LIN {X 0,Y 305.408,Z 165.44,A -85,B 0,C 180,E1 -15880.59,E2 -15880.59} C_VEL
LIN {X 0,Y 305.42,Z 165.439,A -85,B 0,C 180,E1 -15883.657,E2 -15883.657} C_VEL
LIN {X 0,Y 305.434,Z 165.438,A -85,B 0,C 180,E1 -15887.419,E2 -15887.419} C_VEL
LIN {X 0,Y 305.46,Z 165.434,A -85,B 0,C 180,E1 -15891.596,E2 -15891.596} C_VEL
LIN {X 0,Y 305.462,Z 165.438,A -85,B 0,C 180,E1 -15894.887,E2 -15894.887} C_VEL
LIN {X 0,Y 305.446,Z 165.457,A -85,B 0,C 180,E1 -15898.262,E2 -15898.262} C_VEL
LIN {X 0,Y 308.056,Z 177.958,A -85,B 0,C 180,E1 -15902.116,E2 -15902.116} C_VEL
LIN {X 0,Y 309.424,Z 185.81,A -85,B 0,C 180,E1 -15904.434,E2 -15904.434} C_VEL
LIN {X 0,Y 309.211,Z 188.563,A -85,B 0,C 180,E1 -15905.192,E2 -15905.192} C_VEL
LIN {X 0,Y 314.924,Z 228.362,A -85,B 0,C 180,E1 -15906.653,E2 -15906.653} C_VEL
LIN {X 0,Y 313.069,Z 297.497,A -85,B 0,C 180,E1 -15908.433,E2 -15908.433} C_VEL
LIN {X 0,Y 312.295,Z 311.547,A -85,B 0,C 180,E1 -15909.068,E2 -15909.068} C_VEL
LIN {X 0,Y 311.224,Z 323.574,A -85,B 0,C 180,E1 -15909.857,E2 -15909.857} C_VEL
LIN {X 0,Y 310.032,Z 336.146,A -85,B 0,C 180,E1 -15910.982,E2 -15910.982} C_VEL
LIN {X 0,Y 308.666,Z 347.394,A -85,B 0,C 180,E1 -15912.27,E2 -15912.27} C_VEL
LIN {X 0,Y 307.454,Z 358.217,A -85,B 0,C 180,E1 -15913.852,E2 -15913.852} C_VEL
LIN {X 0,Y 306.459,Z 366.753,A -85,B 0,C 180,E1 -15915.389,E2 -15915.389} C_VEL
LIN {X 0,Y 305.37,Z 375.712,A -85,B 0,C 180,E1 -15917.371,E2 -15917.371} C_VEL
LIN {X 0,Y 304.591,Z 382.844,A -85,B 0,C 180,E1 -15919.363,E2 -15919.363} C_VEL
LIN {X 0,Y 304.06,Z 388.526,A -85,B 0,C 180,E1 -15921.359,E2 -15921.359} C_VEL
LIN {X 0,Y 303.758,Z 392.963,A -85,B 0,C 180,E1 -15923.357,E2 -15923.357} C_VEL
LIN {X 0,Y 303.668,Z 395.298,A -85,B 0,C 180,E1 -15924.688,E2 -15924.688} C_VEL
LIN {X 0,Y 303.634,Z 397.179,A -85,B 0,C 180,E1 -15926.018,E2 -15926.018} C_VEL
LIN {X 0,Y 303.608,Z 398.571,A -85,B 0,C 180,E1 -15927.346,E2 -15927.346} C_VEL
LIN {X 0,Y 303.576,Z 399.548,A -85,B 0,C 180,E1 -15928.673,E2 -15928.673} C_VEL
LIN {X 0,Y 303.605,Z 400.123,A -85,B 0,C 180,E1 -15930,E2 -15930} C_VEL
LIN {X 0,Y 303.566,Z 400.276,A -85,B 0,C 180,E1 -15931.326,E2 -15931.326} C_VEL
LIN {X 0,Y 303.602,Z 399.989,A -85,B 0,C 180,E1 -15932.653,E2 -15932.653} C_VEL
LIN {X 0,Y 303.592,Z 399.306,A -85,B 0,C 180,E1 -15933.982,E2 -15933.982} C_VEL
LIN {X 0,Y 303.627,Z 398.001,A -85,B 0,C 180,E1 -15935.544,E2 -15935.544} C_VEL
LIN {X 0,Y 304.004,Z 394.748,A -85,B 0,C 180,E1 -15937.973,E2 -15937.973} C_VEL
LIN {X 0,Y 304.538,Z 390.959,A -85,B 0,C 180,E1 -15939.967,E2 -15939.967} C_VEL
LIN {X 0,Y 305.368,Z 386.046,A -85,B 0,C 180,E1 -15941.954,E2 -15941.954} C_VEL
LIN {X 0,Y 306.544,Z 379.882,A -85,B 0,C 180,E1 -15943.929,E2 -15943.929} C_VEL
LIN {X 0,Y 308.159,Z 372.25,A -85,B 0,C 180,E1 -15945.883,E2 -15945.883} C_VEL
LIN {X 0,Y 309.396,Z 364.671,A -85,B 0,C 180,E1 -15947.481,E2 -15947.481} C_VEL
LIN {X 0,Y 311.169,Z 355.095,A -85,B 0,C 180,E1 -15949.116,E2 -15949.116} C_VEL
LIN {X 0,Y 313.044,Z 344.695,A -85,B 0,C 180,E1 -15950.535,E2 -15950.535} C_VEL
LIN {X 0,Y 314.841,Z 333.237,A -85,B 0,C 180,E1 -15951.783,E2 -15951.783} C_VEL
LIN {X 0,Y 316.432,Z 321.299,A -85,B 0,C 180,E1 -15952.785,E2 -15952.785} C_VEL
LIN {X 0,Y 317.803,Z 308.332,A -85,B 0,C 180,E1 -15953.586,E2 -15953.586} C_VEL
LIN {X 0,Y 318.869,Z 294.721,A -85,B 0,C 180,E1 -15954.149,E2 -15954.149} C_VEL
LIN {X 0,Y 321.21,Z 229.462,A -85,B 0,C 180,E1 -15955.868,E2 -15955.868} C_VEL
LIN {X 0,Y 318.444,Z 211.613,A -85,B 0,C 180,E1 -15956.729,E2 -15956.729} C_VEL
LIN {X 0,Y 315.326,Z 197.331,A -85,B 0,C 180,E1 -15957.545,E2 -15957.545} C_VEL
LIN {X 0,Y 310.558,Z 186.54,A -85,B 0,C 180,E1 -15958.519,E2 -15958.519} C_VEL
LIN {X 0,Y 308.899,Z 178.602,A -85,B 0,C 180,E1 -15961.194,E2 -15961.194} C_VEL
LIN {X 0,Y 306.662,Z 169.805,A -85,B 0,C 180,E1 -15964.407,E2 -15964.407} C_VEL
LIN {X 0,Y 305.483,Z 165.436,A -85,B 0,C 180,E1 -15966.139,E2 -15966.139} C_VEL
LIN {X 0,Y 305.408,Z 165.445,A -85,B 0,C 180,E1 -15970.114,E2 -15970.114} C_VEL
LIN {X 0,Y 305.418,Z 165.446,A -85,B 0,C 180,E1 -15973.655,E2 -15973.655} C_VEL
LIN {X 0,Y 305.431,Z 165.435,A -85,B 0,C 180,E1 -15977.418,E2 -15977.418} C_VEL
LIN {X 0,Y 305.438,Z 165.439,A -85,B 0,C 180,E1 -15981.591,E2 -15981.591} C_VEL
LIN {X 0,Y 305.458,Z 165.437,A -85,B 0,C 180,E1 -15984.886,E2 -15984.886} C_VEL
LIN {X 0,Y 305.438,Z 165.438,A -85,B 0,C 180,E1 -15988.358,E2 -15988.358} C_VEL
LIN {X 0,Y 305.459,Z 165.432,A -85,B 0,C 180,E1 -15991.107,E2 -15991.107} C_VEL
LIN {X 0,Y 305.474,Z 165.424,A -85,B 0,C 180,E1 -15994.078,E2 -15994.078} C_VEL
LIN {X 0,Y 305.452,Z 165.431,A -85,B 0,C 180,E1 -15998.399,E2 -15998.399} C_VEL
LIN {X 0,Y 305.494,Z 165.421,A -85,B 0,C 180,E1 -16001.211,E2 -16001.211} C_VEL
LIN {X 0,Y 305.573,Z 165.414,A -85,B 0,C 180,E1 -16005.345,E2 -16005.345} C_VEL
LIN {X 0,Y 305.617,Z 165.413,A -85,B 0,C 180,E1 -16009.398,E2 -16009.398} C_VEL
LIN {X 0,Y 305.74,Z 165.394,A -85,B 0,C 180,E1 -16012.072,E2 -16012.072} C_VEL
LIN {X 0,Y 305.648,Z 165.405,A -85,B 0,C 180,E1 -16014.722,E2 -16014.722} C_VEL
LIN {X 0,Y 305.928,Z 165.375,A -85,B 0,C 180,E1 -16018.683,E2 -16018.683} C_VEL
LIN {X 0,Y 305.928,Z 165.374,A -85,B 0,C 180,E1 -16021.316,E2 -16021.316} C_VEL
LIN {X 0,Y 305.777,Z 165.398,A -85,B 0,C 180,E1 -16026.598,E2 -16026.598} C_VEL
LIN {X 0,Y 305.688,Z 165.41,A -85,B 0,C 180,E1 -16029.261,E2 -16029.261} C_VEL
LIN {X 0,Y 305.626,Z 165.55,A -85,B 0,C 180,E1 -16031.944,E2 -16031.944} C_VEL
LIN {X 0,Y 307.793,Z 173.872,A -85,B 0,C 180,E1 -16035.181,E2 -16035.181} C_VEL
LIN {X 0,Y 315.177,Z 188.448,A -85,B 0,C 180,E1 -16036.629,E2 -16036.629} C_VEL
LIN {X 0,Y 321.1,Z 202.216,A -85,B 0,C 180,E1 -16037.761,E2 -16037.761} C_VEL
LIN {X 0,Y 322.097,Z 207.438,A -85,B 0,C 180,E1 -16038.033,E2 -16038.033} C_VEL
LIN {X 0,Y 319.132,Z 281.719,A -85,B 0,C 180,E1 -16039.983,E2 -16039.983} C_VEL
LIN {X 0,Y 318.191,Z 294.602,A -85,B 0,C 180,E1 -16040.555,E2 -16040.555} C_VEL
LIN {X 0,Y 317.006,Z 307.445,A -85,B 0,C 180,E1 -16041.39,E2 -16041.39} C_VEL
LIN {X 0,Y 315.544,Z 319.205,A -85,B 0,C 180,E1 -16042.421,E2 -16042.421} C_VEL
LIN {X 0,Y 314.01,Z 329.384,A -85,B 0,C 180,E1 -16043.549,E2 -16043.549} C_VEL
LIN {X 0,Y 312.228,Z 339.663,A -85,B 0,C 180,E1 -16044.963,E2 -16044.963} C_VEL
LIN {X 0,Y 310.555,Z 348.97,A -85,B 0,C 180,E1 -16046.559,E2 -16046.559} C_VEL
LIN {X 0,Y 308.735,Z 358.223,A -85,B 0,C 180,E1 -16048.557,E2 -16048.557} C_VEL
LIN {X 0,Y 307.18,Z 365.75,A -85,B 0,C 180,E1 -16050.601,E2 -16050.601} C_VEL
LIN {X 0,Y 305.96,Z 371.708,A -85,B 0,C 180,E1 -16052.669,E2 -16052.669} C_VEL
LIN {X 0,Y 304.868,Z 377.163,A -85,B 0,C 180,E1 -16055.191,E2 -16055.191} C_VEL
LIN {X 0,Y 304.311,Z 379.879,A -85,B 0,C 180,E1 -16056.902,E2 -16056.902} C_VEL
LIN {X 0,Y 303.863,Z 381.909,A -85,B 0,C 180,E1 -16058.643,E2 -16058.643} C_VEL
LIN {X 0,Y 303.576,Z 383.185,A -85,B 0,C 180,E1 -16060.407,E2 -16060.407} C_VEL
LIN {X 0,Y 303.368,Z 383.757,A -85,B 0,C 180,E1 -16062.208,E2 -16062.208} C_VEL
LIN {X 0,Y 303.301,Z 383.572,A -85,B 0,C 180,E1 -16064.085,E2 -16064.085} C_VEL
LIN {X 0,Y 303.365,Z 382.564,A -85,B 0,C 180,E1 -16065.974,E2 -16065.974} C_VEL
LIN {X 0,Y 303.533,Z 380.734,A -85,B 0,C 180,E1 -16067.821,E2 -16067.821} C_VEL
LIN {X 0,Y 303.8,Z 377.908,A -85,B 0,C 180,E1 -16069.765,E2 -16069.765} C_VEL
LIN {X 0,Y 304.26,Z 373.976,A -85,B 0,C 180,E1 -16071.753,E2 -16071.753} C_VEL
LIN {X 0,Y 304.811,Z 368.708,A -85,B 0,C 180,E1 -16073.802,E2 -16073.802} C_VEL
LIN {X 0,Y 305.595,Z 361.864,A -85,B 0,C 180,E1 -16075.884,E2 -16075.884} C_VEL
LIN {X 0,Y 306.663,Z 353.083,A -85,B 0,C 180,E1 -16077.989,E2 -16077.989} C_VEL
LIN {X 0,Y 307.765,Z 344.443,A -85,B 0,C 180,E1 -16079.654,E2 -16079.654} C_VEL
LIN {X 0,Y 308.949,Z 333.974,A -85,B 0,C 180,E1 -16081.279,E2 -16081.279} C_VEL
LIN {X 0,Y 310.201,Z 322.827,A -85,B 0,C 180,E1 -16082.658,E2 -16082.658} C_VEL
LIN {X 0,Y 311.315,Z 310.616,A -85,B 0,C 180,E1 -16083.842,E2 -16083.842} C_VEL
LIN {X 0,Y 312.329,Z 297.638,A -85,B 0,C 180,E1 -16084.778,E2 -16084.778} C_VEL
LIN {X 0,Y 313.018,Z 284.837,A -85,B 0,C 180,E1 -16085.436,E2 -16085.436} C_VEL
LIN {X 0,Y 313.553,Z 268.917,A -85,B 0,C 180,E1 -16085.921,E2 -16085.921} C_VEL
LIN {X 0,Y 315.327,Z 203.407,A -85,B 0,C 180,E1 -16087.573,E2 -16087.573} C_VEL
LIN {X 0,Y 312.589,Z 189.103,A -85,B 0,C 180,E1 -16088.139,E2 -16088.139} C_VEL
LIN {X 0,Y 306.9,Z 172.553,A -85,B 0,C 180,E1 -16088.991,E2 -16088.991} C_VEL
LIN {X 0,Y 305.545,Z 165.426,A -85,B 0,C 180,E1 -16091.389,E2 -16091.389} C_VEL
LIN {X 0,Y 305.575,Z 165.42,A -85,B 0,C 180,E1 -16095.346,E2 -16095.346} C_VEL
LIN {X 0,Y 305.619,Z 165.413,A -85,B 0,C 180,E1 -16099.399,E2 -16099.399} C_VEL
LIN {X 0,Y 305.743,Z 165.401,A -85,B 0,C 180,E1 -16102.073,E2 -16102.073} C_VEL
LIN {X 0,Y 305.653,Z 165.41,A -85,B 0,C 180,E1 -16104.723,E2 -16104.723} C_VEL
LIN {X 0,Y 305.931,Z 165.376,A -85,B 0,C 180,E1 -16108.684,E2 -16108.684} C_VEL
LIN {X 0,Y 305.93,Z 165.375,A -85,B 0,C 180,E1 -16111.317,E2 -16111.317} C_VEL
LIN {X 0,Y 305.781,Z 165.394,A -85,B 0,C 180,E1 -16116.599,E2 -16116.599} C_VEL
LIN {X 0,Y 305.691,Z 165.405,A -85,B 0,C 180,E1 -16119.261,E2 -16119.261} C_VEL
LIN {X 0,Y 305.566,Z 165.421,A -85,B 0,C 180,E1 -16123.297,E2 -16123.297} C_VEL
LIN {X 0,Y 305.508,Z 165.429,A -85,B 0,C 180,E1 -16126.025,E2 -16126.025} C_VEL
LIN {X 0,Y 305.472,Z 165.432,A -85,B 0,C 180,E1 -16130.188,E2 -16130.188} C_VEL
LIN {X 0,Y 305.435,Z 165.436,A -85,B 0,C 180,E1 -16134.467,E2 -16134.467} C_VEL
LIN {X 0,Y 305.437,Z 165.44,A -85,B 0,C 180,E1 -16137.399,E2 -16137.399} C_VEL
LIN {X 0,Y 305.413,Z 165.438,A -85,B 0,C 180,E1 -16140.414,E2 -16140.414} C_VEL
LIN {X 0,Y 305.461,Z 165.432,A -85,B 0,C 180,E1 -16144.078,E2 -16144.078} C_VEL
LIN {X 0,Y 305.449,Z 165.435,A -85,B 0,C 180,E1 -16146.743,E2 -16146.743} C_VEL
LIN {X 0,Y 305.405,Z 165.44,A -85,B 0,C 180,E1 -16150.59,E2 -16150.59} C_VEL
LIN {X 0,Y 305.416,Z 165.437,A -85,B 0,C 180,E1 -16153.656,E2 -16153.656} C_VEL
LIN {X 0,Y 305.43,Z 165.438,A -85,B 0,C 180,E1 -16157.419,E2 -16157.419} C_VEL
LIN {X 0,Y 305.455,Z 165.434,A -85,B 0,C 180,E1 -16161.595,E2 -16161.595} C_VEL
LIN {X 0,Y 305.439,Z 165.435,A -85,B 0,C 180,E1 -16163.128,E2 -16163.128} C_VEL
LIN {X 0,Y 304.826,Z 165.519,A -85,B 0,C 180,E1 -16164.228,E2 -16164.228} C_VEL
LIN {X 0,Y 301.99,Z 165.879,A -85,B 0,C 180,E1 -16166.019,E2 -16166.019} C_VEL
LIN {X 0,Y 299.537,Z 166.181,A -85,B 0,C 180,E1 -16167.471,E2 -16167.471} C_VEL
LIN {X 0,Y 298.46,Z 166.308,A -85,B 0,C 180,E1 -16168.596,E2 -16168.596} C_VEL
LIN {X 0,Y 298.363,Z 166.317,A -85,B 0,C 180,E1 -16168.978,E2 -16168.978} C_VEL
LIN {X 0,Y 298.404,Z 166.311,A -85,B 0,C 180,E1 -16171.899,E2 -16171.899} C_VEL
LIN {X 0,Y 298.408,Z 166.314,A -85,B 0,C 180,E1 -16174.918,E2 -16174.918} C_VEL
LIN {X 0,Y 298.386,Z 166.313,A -85,B 0,C 180,E1 -16177.862,E2 -16177.862} C_VEL
LIN {X 0,Y 298.448,Z 166.304,A -85,B 0,C 180,E1 -16180.751,E2 -16180.751} C_VEL
LIN {X 0,Y 298.506,Z 166.298,A -85,B 0,C 180,E1 -16184.991,E2 -16184.991} C_VEL
LIN {X 0,Y 298.576,Z 166.29,A -85,B 0,C 180,E1 -16189.147,E2 -16189.147} C_VEL
LIN {X 0,Y 298.68,Z 166.278,A -85,B 0,C 180,E1 -16191.884,E2 -16191.884} C_VEL
LIN {X 0,Y 298.62,Z 166.282,A -85,B 0,C 180,E1 -16194.599,E2 -16194.599} C_VEL
LIN {X 0,Y 298.897,Z 166.25,A -85,B 0,C 180,E1 -16198.653,E2 -16198.653} C_VEL
LIN {X 0,Y 298.897,Z 166.25,A -85,B 0,C 180,E1 -16201.348,E2 -16201.348} C_VEL
LIN {X 0,Y 298.728,Z 166.268,A -85,B 0,C 180,E1 -16206.756,E2 -16206.756} C_VEL
LIN {X 0,Y 298.614,Z 166.287,A -85,B 0,C 180,E1 -16209.483,E2 -16209.483} C_VEL
LIN {X 0,Y 298.519,Z 166.301,A -85,B 0,C 180,E1 -16213.617,E2 -16213.617} C_VEL
LIN {X 0,Y 298.443,Z 166.305,A -85,B 0,C 180,E1 -16216.415,E2 -16216.415} C_VEL
LIN {X 0,Y 298.426,Z 166.314,A -85,B 0,C 180,E1 -16219.61,E2 -16219.61} C_VEL
LIN {X 0,Y 298.379,Z 166.318,A -85,B 0,C 180,E1 -16223.605,E2 -16223.605} C_VEL
LIN {X 0,Y 298.399,Z 166.313,A -85,B 0,C 180,E1 -16226.584,E2 -16226.584} C_VEL
LIN {X 0,Y 298.355,Z 166.321,A -85,B 0,C 180,E1 -16229.649,E2 -16229.649} C_VEL
LIN {X 0,Y 298.391,Z 166.312,A -85,B 0,C 180,E1 -16232.801,E2 -16232.801} C_VEL
LIN {X 0,Y 298.426,Z 166.31,A -85,B 0,C 180,E1 -16236.803,E2 -16236.803} C_VEL
LIN {X 0,Y 298.373,Z 166.318,A -85,B 0,C 180,E1 -16239.493,E2 -16239.493} C_VEL
LIN {X 0,Y 298.369,Z 166.321,A -85,B 0,C 180,E1 -16243.098,E2 -16243.098} C_VEL
LIN {X 0,Y 298.37,Z 166.321,A -85,B 0,C 180,E1 -16246.915,E2 -16246.915} C_VEL
LIN {X 0,Y 298.385,Z 166.319,A -85,B 0,C 180,E1 -16251.012,E2 -16251.012} C_VEL
LIN {X 0,Y 298.405,Z 166.313,A -85,B 0,C 180,E1 -16253.929,E2 -16253.929} C_VEL
LIN {X 0,Y 298.421,Z 166.42,A -85,B 0,C 180,E1 -16257.932,E2 -16257.932} C_VEL
LIN {X 0,Y 300.947,Z 178.583,A -85,B 0,C 180,E1 -16261.778,E2 -16261.778} C_VEL
LIN {X 0,Y 302.396,Z 186.453,A -85,B 0,C 180,E1 -16264.164,E2 -16264.164} C_VEL
LIN {X 0,Y 302.387,Z 188.388,A -85,B 0,C 180,E1 -16264.72,E2 -16264.72} C_VEL
LIN {X 0,Y 308.176,Z 228.777,A -85,B 0,C 180,E1 -16266.25,E2 -16266.25} C_VEL
LIN {X 0,Y 306.271,Z 297.409,A -85,B 0,C 180,E1 -16268.062,E2 -16268.062} C_VEL
LIN {X 0,Y 305.454,Z 311.406,A -85,B 0,C 180,E1 -16268.709,E2 -16268.709} C_VEL
LIN {X 0,Y 304.33,Z 323.913,A -85,B 0,C 180,E1 -16269.556,E2 -16269.556} C_VEL
LIN {X 0,Y 303.105,Z 336.378,A -85,B 0,C 180,E1 -16270.706,E2 -16270.706} C_VEL
LIN {X 0,Y 301.703,Z 347.545,A -85,B 0,C 180,E1 -16272.022,E2 -16272.022} C_VEL
LIN {X 0,Y 300.642,Z 357.023,A -85,B 0,C 180,E1 -16273.426,E2 -16273.426} C_VEL
LIN {X 0,Y 299.563,Z 365.961,A -85,B 0,C 180,E1 -16275.044,E2 -16275.044} C_VEL
LIN {X 0,Y 298.418,Z 375.024,A -85,B 0,C 180,E1 -16277.072,E2 -16277.072} C_VEL
LIN {X 0,Y 297.571,Z 382.282,A -85,B 0,C 180,E1 -16279.109,E2 -16279.109} C_VEL
LIN {X 0,Y 297.012,Z 388.04,A -85,B 0,C 180,E1 -16281.152,E2 -16281.152} C_VEL
LIN {X 0,Y 296.698,Z 392.547,A -85,B 0,C 180,E1 -16283.198,E2 -16283.198} C_VEL
LIN {X 0,Y 296.602,Z 394.914,A -85,B 0,C 180,E1 -16284.561,E2 -16284.561} C_VEL
LIN {X 0,Y 296.534,Z 396.835,A -85,B 0,C 180,E1 -16285.923,E2 -16285.923} C_VEL
LIN {X 0,Y 296.535,Z 398.277,A -85,B 0,C 180,E1 -16287.283,E2 -16287.283} C_VEL
LIN {X 0,Y 296.496,Z 399.282,A -85,B 0,C 180,E1 -16288.642,E2 -16288.642} C_VEL
LIN {X 0,Y 296.52,Z 399.885,A -85,B 0,C 180,E1 -16290,E2 -16290} C_VEL
LIN {X 0,Y 296.486,Z 400.081,A -85,B 0,C 180,E1 -16291.358,E2 -16291.358} C_VEL
LIN {X 0,Y 296.526,Z 399.831,A -85,B 0,C 180,E1 -16292.717,E2 -16292.717} C_VEL
LIN {X 0,Y 296.493,Z 399.172,A -85,B 0,C 180,E1 -16294.078,E2 -16294.078} C_VEL
LIN {X 0,Y 296.548,Z 398.058,A -85,B 0,C 180,E1 -16295.508,E2 -16295.508} C_VEL
LIN {X 0,Y 296.69,Z 396.655,A -85,B 0,C 180,E1 -16296.802,E2 -16296.802} C_VEL
LIN {X 0,Y 297.126,Z 393.616,A -85,B 0,C 180,E1 -16298.844,E2 -16298.844} C_VEL
LIN {X 0,Y 297.788,Z 389.537,A -85,B 0,C 180,E1 -16300.883,E2 -16300.883} C_VEL
LIN {X 0,Y 298.955,Z 383.297,A -85,B 0,C 180,E1 -16303.25,E2 -16303.25} C_VEL
LIN {X 0,Y 300.451,Z 376.51,A -85,B 0,C 180,E1 -16305.257,E2 -16305.257} C_VEL
LIN {X 0,Y 301.704,Z 370.268,A -85,B 0,C 180,E1 -16306.78,E2 -16306.78} C_VEL
LIN {X 0,Y 303.298,Z 361.562,A -85,B 0,C 180,E1 -16308.544,E2 -16308.544} C_VEL
LIN {X 0,Y 305.329,Z 351.35,A -85,B 0,C 180,E1 -16310.198,E2 -16310.198} C_VEL
LIN {X 0,Y 307.364,Z 340.093,A -85,B 0,C 180,E1 -16311.635,E2 -16311.635} C_VEL
LIN {X 0,Y 309.281,Z 327.482,A -85,B 0,C 180,E1 -16312.901,E2 -16312.901} C_VEL
LIN {X 0,Y 310.914,Z 314.905,A -85,B 0,C 180,E1 -16313.831,E2 -16313.831} C_VEL
LIN {X 0,Y 312.293,Z 301,A -85,B 0,C 180,E1 -16314.558,E2 -16314.558} C_VEL
LIN {X 0,Y 313.097,Z 286.646,A -85,B 0,C 180,E1 -16315.022,E2 -16315.022} C_VEL
LIN {X 0,Y 315.149,Z 230.45,A -85,B 0,C 180,E1 -16316.523,E2 -16316.523} C_VEL
LIN {X 0,Y 312.435,Z 212.921,A -85,B 0,C 180,E1 -16317.399,E2 -16317.399} C_VEL
LIN {X 0,Y 309.852,Z 200.583,A -85,B 0,C 180,E1 -16318.13,E2 -16318.13} C_VEL
LIN {X 0,Y 303.398,Z 186.182,A -85,B 0,C 180,E1 -16319.529,E2 -16319.529} C_VEL
LIN {X 0,Y 301.559,Z 178.102,A -85,B 0,C 180,E1 -16322.413,E2 -16322.413} C_VEL
LIN {X 0,Y 299.161,Z 168.943,A -85,B 0,C 180,E1 -16325.965,E2 -16325.965} C_VEL
LIN {X 0,Y 298.385,Z 166.318,A -85,B 0,C 180,E1 -16327.088,E2 -16327.088} C_VEL
LIN {X 0,Y 298.346,Z 166.328,A -85,B 0,C 180,E1 -16331.267,E2 -16331.267} C_VEL
LIN {X 0,Y 298.353,Z 166.32,A -85,B 0,C 180,E1 -16335.034,E2 -16335.034} C_VEL
LIN {X 0,Y 298.345,Z 166.324,A -85,B 0,C 180,E1 -16338.92,E2 -16338.92} C_VEL
LIN {X 0,Y 298.384,Z 166.318,A -85,B 0,C 180,E1 -16342.237,E2 -16342.237} C_VEL
LIN {X 0,Y 298.405,Z 166.312,A -85,B 0,C 180,E1 -16345.58,E2 -16345.58} C_VEL
LIN {X 0,Y 298.369,Z 166.317,A -85,B 0,C 180,E1 -16348.788,E2 -16348.788} C_VEL
LIN {X 0,Y 298.399,Z 166.314,A -85,B 0,C 180,E1 -16351.897,E2 -16351.897} C_VEL
LIN {X 0,Y 298.416,Z 166.311,A -85,B 0,C 180,E1 -16354.917,E2 -16354.917} C_VEL
LIN {X 0,Y 298.385,Z 166.307,A -85,B 0,C 180,E1 -16357.86,E2 -16357.86} C_VEL
LIN {X 0,Y 298.447,Z 166.3,A -85,B 0,C 180,E1 -16360.75,E2 -16360.75} C_VEL
LIN {X 0,Y 298.505,Z 166.293,A -85,B 0,C 180,E1 -16364.99,E2 -16364.99} C_VEL
LIN {X 0,Y 298.575,Z 166.289,A -85,B 0,C 180,E1 -16369.145,E2 -16369.145} C_VEL
LIN {X 0,Y 298.691,Z 166.272,A -85,B 0,C 180,E1 -16371.884,E2 -16371.884} C_VEL
LIN {X 0,Y 298.618,Z 166.281,A -85,B 0,C 180,E1 -16374.598,E2 -16374.598} C_VEL
LIN {X 0,Y 298.896,Z 166.251,A -85,B 0,C 180,E1 -16378.652,E2 -16378.652} C_VEL
LIN {X 0,Y 298.896,Z 166.25,A -85,B 0,C 180,E1 -16381.347,E2 -16381.347} C_VEL
LIN {X 0,Y 298.726,Z 166.276,A -85,B 0,C 180,E1 -16386.755,E2 -16386.755} C_VEL
LIN {X 0,Y 298.618,Z 166.29,A -85,B 0,C 180,E1 -16389.482,E2 -16389.482} C_VEL
LIN {X 0,Y 298.615,Z 166.457,A -85,B 0,C 180,E1 -16391.024,E2 -16391.024} C_VEL
LIN {X 0,Y 300.639,Z 174.15,A -85,B 0,C 180,E1 -16394.165,E2 -16394.165} C_VEL
LIN {X 0,Y 308.786,Z 189.813,A -85,B 0,C 180,E1 -16395.85,E2 -16395.85} C_VEL
LIN {X 0,Y 314.879,Z 203.614,A -85,B 0,C 180,E1 -16397.076,E2 -16397.076} C_VEL
LIN {X 0,Y 315.859,Z 207.46,A -85,B 0,C 180,E1 -16397.313,E2 -16397.313} C_VEL
LIN {X 0,Y 316.009,Z 210.613,A -85,B 0,C 180,E1 -16397.43,E2 -16397.43} C_VEL
LIN {X 0,Y 313.021,Z 281.822,A -85,B 0,C 180,E1 -16399.334,E2 -16399.334} C_VEL
LIN {X 0,Y 311.985,Z 294.897,A -85,B 0,C 180,E1 -16399.92,E2 -16399.92} C_VEL
LIN {X 0,Y 310.743,Z 307.8,A -85,B 0,C 180,E1 -16400.781,E2 -16400.781} C_VEL
LIN {X 0,Y 309.136,Z 319.952,A -85,B 0,C 180,E1 -16401.877,E2 -16401.877} C_VEL
LIN {X 0,Y 307.412,Z 330.743,A -85,B 0,C 180,E1 -16403.12,E2 -16403.12} C_VEL
LIN {X 0,Y 305.457,Z 341.319,A -85,B 0,C 180,E1 -16404.646,E2 -16404.646} C_VEL
LIN {X 0,Y 303.546,Z 351.257,A -85,B 0,C 180,E1 -16406.467,E2 -16406.467} C_VEL
LIN {X 0,Y 301.947,Z 358.817,A -85,B 0,C 180,E1 -16408.175,E2 -16408.175} C_VEL
LIN {X 0,Y 300.469,Z 365.637,A -85,B 0,C 180,E1 -16410.07,E2 -16410.07} C_VEL
LIN {X 0,Y 299.116,Z 371.822,A -85,B 0,C 180,E1 -16412.238,E2 -16412.238} C_VEL
LIN {X 0,Y 298.063,Z 376.646,A -85,B 0,C 180,E1 -16414.464,E2 -16414.464} C_VEL
LIN {X 0,Y 297.327,Z 379.958,A -85,B 0,C 180,E1 -16416.52,E2 -16416.52} C_VEL
LIN {X 0,Y 296.8,Z 382.282,A -85,B 0,C 180,E1 -16418.611,E2 -16418.611} C_VEL
LIN {X 0,Y 296.461,Z 383.607,A -85,B 0,C 180,E1 -16420.66,E2 -16420.66} C_VEL
LIN {X 0,Y 296.233,Z 384.01,A -85,B 0,C 180,E1 -16422.655,E2 -16422.655} C_VEL
LIN {X 0,Y 296.233,Z 383.102,A -85,B 0,C 180,E1 -16425.376,E2 -16425.376} C_VEL
LIN {X 0,Y 296.38,Z 381.468,A -85,B 0,C 180,E1 -16427.314,E2 -16427.314} C_VEL
LIN {X 0,Y 296.632,Z 378.886,A -85,B 0,C 180,E1 -16429.302,E2 -16429.302} C_VEL
LIN {X 0,Y 297.067,Z 375.236,A -85,B 0,C 180,E1 -16431.325,E2 -16431.325} C_VEL
LIN {X 0,Y 297.596,Z 370.283,A -85,B 0,C 180,E1 -16433.411,E2 -16433.411} C_VEL
LIN {X 0,Y 298.286,Z 363.737,A -85,B 0,C 180,E1 -16435.566,E2 -16435.566} C_VEL
LIN {X 0,Y 299.372,Z 355.582,A -85,B 0,C 180,E1 -16437.684,E2 -16437.684} C_VEL
LIN {X 0,Y 300.498,Z 346.961,A -85,B 0,C 180,E1 -16439.47,E2 -16439.47} C_VEL
LIN {X 0,Y 301.755,Z 336.567,A -85,B 0,C 180,E1 -16441.213,E2 -16441.213} C_VEL
LIN {X 0,Y 302.907,Z 326.732,A -85,B 0,C 180,E1 -16442.54,E2 -16442.54} C_VEL
LIN {X 0,Y 304.034,Z 315.383,A -85,B 0,C 180,E1 -16443.763,E2 -16443.763} C_VEL
LIN {X 0,Y 305.149,Z 303.096,A -85,B 0,C 180,E1 -16444.782,E2 -16444.782} C_VEL
LIN {X 0,Y 305.954,Z 290.042,A -85,B 0,C 180,E1 -16445.577,E2 -16445.577} C_VEL
LIN {X 0,Y 306.625,Z 276.064,A -85,B 0,C 180,E1 -16446.115,E2 -16446.115} C_VEL
LIN {X 0,Y 308.685,Z 204.716,A -85,B 0,C 180,E1 -16447.96,E2 -16447.96} C_VEL
LIN {X 0,Y 306.185,Z 191.454,A -85,B 0,C 180,E1 -16448.498,E2 -16448.498} C_VEL
LIN {X 0,Y 299.727,Z 172.695,A -85,B 0,C 180,E1 -16449.511,E2 -16449.511} C_VEL
LIN {X 0,Y 298.489,Z 166.304,A -85,B 0,C 180,E1 -16451.733,E2 -16451.733} C_VEL
LIN {X 0,Y 298.507,Z 166.302,A -85,B 0,C 180,E1 -16454.991,E2 -16454.991} C_VEL
LIN {X 0,Y 298.577,Z 166.291,A -85,B 0,C 180,E1 -16459.146,E2 -16459.146} C_VEL
LIN {X 0,Y 298.694,Z 166.277,A -85,B 0,C 180,E1 -16461.885,E2 -16461.885} C_VEL
LIN {X 0,Y 298.623,Z 166.287,A -85,B 0,C 180,E1 -16464.599,E2 -16464.599} C_VEL
LIN {X 0,Y 298.899,Z 166.252,A -85,B 0,C 180,E1 -16468.653,E2 -16468.653} C_VEL
LIN {X 0,Y 298.898,Z 166.252,A -85,B 0,C 180,E1 -16471.348,E2 -16471.348} C_VEL
LIN {X 0,Y 298.73,Z 166.272,A -85,B 0,C 180,E1 -16476.756,E2 -16476.756} C_VEL
LIN {X 0,Y 298.622,Z 166.287,A -85,B 0,C 180,E1 -16479.482,E2 -16479.482} C_VEL
LIN {X 0,Y 298.519,Z 166.302,A -85,B 0,C 180,E1 -16483.617,E2 -16483.617} C_VEL
LIN {X 0,Y 298.448,Z 166.307,A -85,B 0,C 180,E1 -16486.414,E2 -16486.414} C_VEL
LIN {X 0,Y 298.428,Z 166.314,A -85,B 0,C 180,E1 -16489.611,E2 -16489.611} C_VEL
LIN {X 0,Y 298.378,Z 166.32,A -85,B 0,C 180,E1 -16493.604,E2 -16493.604} C_VEL
LIN {X 0,Y 298.397,Z 166.313,A -85,B 0,C 180,E1 -16496.583,E2 -16496.583} C_VEL
LIN {X 0,Y 298.353,Z 166.32,A -85,B 0,C 180,E1 -16499.648,E2 -16499.648} C_VEL
LIN {X 0,Y 298.389,Z 166.312,A -85,B 0,C 180,E1 -16502.801,E2 -16502.801} C_VEL
LIN {X 0,Y 298.424,Z 166.311,A -85,B 0,C 180,E1 -16506.803,E2 -16506.803} C_VEL
LIN {X 0,Y 298.369,Z 166.318,A -85,B 0,C 180,E1 -16509.492,E2 -16509.492} C_VEL
LIN {X 0,Y 298.365,Z 166.318,A -85,B 0,C 180,E1 -16513.097,E2 -16513.097} C_VEL
LIN {X 0,Y 298.366,Z 166.319,A -85,B 0,C 180,E1 -16516.915,E2 -16516.915} C_VEL
LIN {X 0,Y 298.38,Z 166.319,A -85,B 0,C 180,E1 -16521.011,E2 -16521.011} C_VEL
LIN {X 0,Y 298.399,Z 166.311,A -85,B 0,C 180,E1 -16523.928,E2 -16523.928} C_VEL
LIN {X 0,Y 298.388,Z 166.312,A -85,B 0,C 180,E1 -16527.2,E2 -16527.2} C_VEL
LIN {X 0,Y 298.363,Z 166.317,A -85,B 0,C 180,E1 -16528.978,E2 -16528.978} C_VEL
LIN {X 0,Y 297.671,Z 166.403,A -85,B 0,C 180,E1 -16530.105,E2 -16530.105} C_VEL
LIN {X 0,Y 294.822,Z 166.758,A -85,B 0,C 180,E1 -16531.942,E2 -16531.942} C_VEL
LIN {X 0,Y 292.421,Z 167.057,A -85,B 0,C 180,E1 -16533.432,E2 -16533.432} C_VEL
LIN {X 0,Y 291.39,Z 167.19,A -85,B 0,C 180,E1 -16534.586,E2 -16534.586} C_VEL
LIN {X 0,Y 291.304,Z 167.194,A -85,B 0,C 180,E1 -16534.977,E2 -16534.977} C_VEL
LIN {X 0,Y 291.337,Z 167.192,A -85,B 0,C 180,E1 -16538.787,E2 -16538.787} C_VEL
LIN {X 0,Y 291.378,Z 167.181,A -85,B 0,C 180,E1 -16541.727,E2 -16541.727} C_VEL
LIN {X 0,Y 291.47,Z 167.177,A -85,B 0,C 180,E1 -16544.683,E2 -16544.683} C_VEL
LIN {X 0,Y 291.522,Z 167.169,A -85,B 0,C 180,E1 -16548.881,E2 -16548.881} C_VEL
LIN {X 0,Y 291.626,Z 167.156,A -85,B 0,C 180,E1 -16551.687,E2 -16551.687} C_VEL
LIN {X 0,Y 291.59,Z 167.158,A -85,B 0,C 180,E1 -16554.468,E2 -16554.468} C_VEL
LIN {X 0,Y 291.864,Z 167.126,A -85,B 0,C 180,E1 -16558.621,E2 -16558.621} C_VEL
LIN {X 0,Y 291.864,Z 167.127,A -85,B 0,C 180,E1 -16561.38,E2 -16561.38} C_VEL
LIN {X 0,Y 291.679,Z 167.146,A -85,B 0,C 180,E1 -16566.92,E2 -16566.92} C_VEL
LIN {X 0,Y 291.56,Z 167.167,A -85,B 0,C 180,E1 -16569.715,E2 -16569.715} C_VEL
LIN {X 0,Y 291.478,Z 167.177,A -85,B 0,C 180,E1 -16573.953,E2 -16573.953} C_VEL
LIN {X 0,Y 291.395,Z 167.182,A -85,B 0,C 180,E1 -16576.824,E2 -16576.824} C_VEL
LIN {X 0,Y 291.389,Z 167.189,A -85,B 0,C 180,E1 -16579.843,E2 -16579.843} C_VEL
LIN {X 0,Y 291.323,Z 167.193,A -85,B 0,C 180,E1 -16584.213,E2 -16584.213} C_VEL
LIN {X 0,Y 291.326,Z 167.198,A -85,B 0,C 180,E1 -16587.282,E2 -16587.282} C_VEL
LIN {X 0,Y 291.3,Z 167.196,A -85,B 0,C 180,E1 -16590.442,E2 -16590.442} C_VEL
LIN {X 0,Y 291.342,Z 167.19,A -85,B 0,C 180,E1 -16593.699,E2 -16593.699} C_VEL
LIN {X 0,Y 291.357,Z 167.194,A -85,B 0,C 180,E1 -16597.25,E2 -16597.25} C_VEL
LIN {X 0,Y 291.299,Z 167.198,A -85,B 0,C 180,E1 -16600.649,E2 -16600.649} C_VEL
LIN {X 0,Y 291.281,Z 167.2,A -85,B 0,C 180,E1 -16604.404,E2 -16604.404} C_VEL
LIN {X 0,Y 291.294,Z 167.199,A -85,B 0,C 180,E1 -16608.412,E2 -16608.412} C_VEL
LIN {X 0,Y 291.334,Z 167.196,A -85,B 0,C 180,E1 -16611.156,E2 -16611.156} C_VEL
LIN {X 0,Y 291.356,Z 167.194,A -85,B 0,C 180,E1 -16614.626,E2 -16614.626} C_VEL
LIN {X 0,Y 291.392,Z 167.335,A -85,B 0,C 180,E1 -16617.583,E2 -16617.583} C_VEL
LIN {X 0,Y 293.856,Z 179.18,A -85,B 0,C 180,E1 -16621.424,E2 -16621.424} C_VEL
LIN {X 0,Y 295.494,Z 188.452,A -85,B 0,C 180,E1 -16624.237,E2 -16624.237} C_VEL
LIN {X 0,Y 301.267,Z 228.083,A -85,B 0,C 180,E1 -16625.787,E2 -16625.787} C_VEL
LIN {X 0,Y 301.32,Z 235.203,A -85,B 0,C 180,E1 -16625.994,E2 -16625.994} C_VEL
LIN {X 0,Y 299.496,Z 297.326,A -85,B 0,C 180,E1 -16627.675,E2 -16627.675} C_VEL
LIN {X 0,Y 298.651,Z 311.273,A -85,B 0,C 180,E1 -16628.336,E2 -16628.336} C_VEL
LIN {X 0,Y 297.564,Z 323.267,A -85,B 0,C 180,E1 -16629.161,E2 -16629.161} C_VEL
LIN {X 0,Y 296.307,Z 335.012,A -85,B 0,C 180,E1 -16630.246,E2 -16630.246} C_VEL
LIN {X 0,Y 294.884,Z 346.401,A -85,B 0,C 180,E1 -16631.592,E2 -16631.592} C_VEL
LIN {X 0,Y 293.665,Z 357.068,A -85,B 0,C 180,E1 -16633.194,E2 -16633.194} C_VEL
LIN {X 0,Y 292.417,Z 366.823,A -85,B 0,C 180,E1 -16635.027,E2 -16635.027} C_VEL
LIN {X 0,Y 291.465,Z 374.334,A -85,B 0,C 180,E1 -16636.758,E2 -16636.758} C_VEL
LIN {X 0,Y 290.533,Z 381.699,A -85,B 0,C 180,E1 -16638.842,E2 -16638.842} C_VEL
LIN {X 0,Y 289.976,Z 387.554,A -85,B 0,C 180,E1 -16640.936,E2 -16640.936} C_VEL
LIN {X 0,Y 289.639,Z 392.13,A -85,B 0,C 180,E1 -16643.031,E2 -16643.031} C_VEL
LIN {X 0,Y 289.519,Z 394.53,A -85,B 0,C 180,E1 -16644.428,E2 -16644.428} C_VEL
LIN {X 0,Y 289.439,Z 396.481,A -85,B 0,C 180,E1 -16645.822,E2 -16645.822} C_VEL
LIN {X 0,Y 289.462,Z 397.983,A -85,B 0,C 180,E1 -16647.216,E2 -16647.216} C_VEL
LIN {X 0,Y 289.417,Z 399.016,A -85,B 0,C 180,E1 -16648.608,E2 -16648.608} C_VEL
LIN {X 0,Y 289.437,Z 399.646,A -85,B 0,C 180,E1 -16650,E2 -16650} C_VEL
LIN {X 0,Y 289.408,Z 399.873,A -85,B 0,C 180,E1 -16651.391,E2 -16651.391} C_VEL
LIN {X 0,Y 289.43,Z 399.673,A -85,B 0,C 180,E1 -16652.783,E2 -16652.783} C_VEL
LIN {X 0,Y 289.478,Z 398.02,A -85,B 0,C 180,E1 -16655.573,E2 -16655.573} C_VEL
LIN {X 0,Y 289.636,Z 396.597,A -85,B 0,C 180,E1 -16656.968,E2 -16656.968} C_VEL
LIN {X 0,Y 290.082,Z 393.617,A -85,B 0,C 180,E1 -16659.06,E2 -16659.06} C_VEL
LIN {X 0,Y 290.801,Z 389.601,A -85,B 0,C 180,E1 -16661.147,E2 -16661.147} C_VEL
LIN {X 0,Y 292.02,Z 383.465,A -85,B 0,C 180,E1 -16663.571,E2 -16663.571} C_VEL
LIN {X 0,Y 293.621,Z 376.752,A -85,B 0,C 180,E1 -16665.621,E2 -16665.621} C_VEL
LIN {X 0,Y 295.097,Z 369.131,A -85,B 0,C 180,E1 -16667.521,E2 -16667.521} C_VEL
LIN {X 0,Y 297.079,Z 360.068,A -85,B 0,C 180,E1 -16669.341,E2 -16669.341} C_VEL
LIN {X 0,Y 298.904,Z 350.928,A -85,B 0,C 180,E1 -16670.831,E2 -16670.831} C_VEL
LIN {X 0,Y 301.109,Z 339.63,A -85,B 0,C 180,E1 -16672.289,E2 -16672.289} C_VEL
LIN {X 0,Y 302.82,Z 328.694,A -85,B 0,C 180,E1 -16673.418,E2 -16673.418} C_VEL
LIN {X 0,Y 304.5,Z 316.708,A -85,B 0,C 180,E1 -16674.365,E2 -16674.365} C_VEL
LIN {X 0,Y 305.951,Z 303.589,A -85,B 0,C 180,E1 -16675.102,E2 -16675.102} C_VEL
LIN {X 0,Y 306.885,Z 289.866,A -85,B 0,C 180,E1 -16675.61,E2 -16675.61} C_VEL
LIN {X 0,Y 309.166,Z 231.503,A -85,B 0,C 180,E1 -16677.203,E2 -16677.203} C_VEL
LIN {X 0,Y 306.466,Z 213.635,A -85,B 0,C 180,E1 -16678.14,E2 -16678.14} C_VEL
LIN {X 0,Y 304.334,Z 203.594,A -85,B 0,C 180,E1 -16678.76,E2 -16678.76} C_VEL
LIN {X 0,Y 298.024,Z 189.846,A -85,B 0,C 180,E1 -16680.14,E2 -16680.14} C_VEL
LIN {X 0,Y 296.248,Z 186.01,A -85,B 0,C 180,E1 -16680.56,E2 -16680.56} C_VEL
LIN {X 0,Y 293.94,Z 176.453,A -85,B 0,C 180,E1 -16684.184,E2 -16684.184} C_VEL
LIN {X 0,Y 291.773,Z 168.876,A -85,B 0,C 180,E1 -16687.356,E2 -16687.356} C_VEL
LIN {X 0,Y 291.323,Z 167.199,A -85,B 0,C 180,E1 -16688.198,E2 -16688.198} C_VEL
LIN {X 0,Y 291.285,Z 167.203,A -85,B 0,C 180,E1 -16692.497,E2 -16692.497} C_VEL
LIN {X 0,Y 291.287,Z 167.205,A -85,B 0,C 180,E1 -16696.37,E2 -16696.37} C_VEL
LIN {X 0,Y 291.354,Z 167.187,A -85,B 0,C 180,E1 -16700.523,E2 -16700.523} C_VEL
LIN {X 0,Y 291.382,Z 167.183,A -85,B 0,C 180,E1 -16702.915,E2 -16702.915} C_VEL
LIN {X 0,Y 291.34,Z 167.187,A -85,B 0,C 180,E1 -16706.3,E2 -16706.3} C_VEL
LIN {X 0,Y 291.334,Z 167.186,A -85,B 0,C 180,E1 -16710.277,E2 -16710.277} C_VEL
LIN {X 0,Y 291.341,Z 167.185,A -85,B 0,C 180,E1 -16714.264,E2 -16714.264} C_VEL
LIN {X 0,Y 291.345,Z 167.183,A -85,B 0,C 180,E1 -16717.296,E2 -16717.296} C_VEL
LIN {X 0,Y 291.38,Z 167.184,A -85,B 0,C 180,E1 -16720.264,E2 -16720.264} C_VEL
LIN {X 0,Y 291.469,Z 167.169,A -85,B 0,C 180,E1 -16724.682,E2 -16724.682} C_VEL
LIN {X 0,Y 291.521,Z 167.165,A -85,B 0,C 180,E1 -16728.879,E2 -16728.879} C_VEL
LIN {X 0,Y 291.645,Z 167.149,A -85,B 0,C 180,E1 -16731.686,E2 -16731.686} C_VEL
LIN {X 0,Y 291.589,Z 167.158,A -85,B 0,C 180,E1 -16734.467,E2 -16734.467} C_VEL
LIN {X 0,Y 291.864,Z 167.126,A -85,B 0,C 180,E1 -16738.62,E2 -16738.62} C_VEL
LIN {X 0,Y 291.863,Z 167.126,A -85,B 0,C 180,E1 -16741.379,E2 -16741.379} C_VEL
LIN {X 0,Y 291.679,Z 167.154,A -85,B 0,C 180,E1 -16746.919,E2 -16746.919} C_VEL
LIN {X 0,Y 291.58,Z 167.289,A -85,B 0,C 180,E1 -16749.976,E2 -16749.976} C_VEL
LIN {X 0,Y 293.607,Z 174.69,A -85,B 0,C 180,E1 -16753.099,E2 -16753.099} C_VEL
LIN {X 0,Y 300.955,Z 188.273,A -85,B 0,C 180,E1 -16754.718,E2 -16754.718} C_VEL
LIN {X 0,Y 307.132,Z 201.342,A -85,B 0,C 180,E1 -16756.014,E2 -16756.014} C_VEL
LIN {X 0,Y 309.856,Z 208.22,A -85,B 0,C 180,E1 -16756.597,E2 -16756.597} C_VEL
LIN {X 0,Y 310.037,Z 211.726,A -85,B 0,C 180,E1 -16756.735,E2 -16756.735} C_VEL
LIN {X 0,Y 306.877,Z 282.62,A -85,B 0,C 180,E1 -16758.683,E2 -16758.683} C_VEL
LIN {X 0,Y 305.817,Z 295.581,A -85,B 0,C 180,E1 -16759.285,E2 -16759.285} C_VEL
LIN {X 0,Y 304.554,Z 308.092,A -85,B 0,C 180,E1 -16760.14,E2 -16760.14} C_VEL
LIN {X 0,Y 302.86,Z 320.241,A -85,B 0,C 180,E1 -16761.255,E2 -16761.255} C_VEL
LIN {X 0,Y 301.139,Z 330.602,A -85,B 0,C 180,E1 -16762.467,E2 -16762.467} C_VEL
LIN {X 0,Y 299.093,Z 341.125,A -85,B 0,C 180,E1 -16763.997,E2 -16763.997} C_VEL
LIN {X 0,Y 297.383,Z 349.574,A -85,B 0,C 180,E1 -16765.532,E2 -16765.532} C_VEL
LIN {X 0,Y 295.465,Z 358.207,A -85,B 0,C 180,E1 -16767.468,E2 -16767.468} C_VEL
LIN {X 0,Y 293.588,Z 366.39,A -85,B 0,C 180,E1 -16769.782,E2 -16769.782} C_VEL
LIN {X 0,Y 292.175,Z 372.316,A -85,B 0,C 180,E1 -16771.95,E2 -16771.95} C_VEL
LIN {X 0,Y 291.291,Z 376.125,A -85,B 0,C 180,E1 -16773.705,E2 -16773.705} C_VEL
LIN {X 0,Y 290.587,Z 379.138,A -85,B 0,C 180,E1 -16775.482,E2 -16775.482} C_VEL
LIN {X 0,Y 290.004,Z 381.467,A -85,B 0,C 180,E1 -16777.29,E2 -16777.29} C_VEL
LIN {X 0,Y 289.603,Z 383.097,A -85,B 0,C 180,E1 -16779.12,E2 -16779.12} C_VEL
LIN {X 0,Y 289.319,Z 384.035,A -85,B 0,C 180,E1 -16781.147,E2 -16781.147} C_VEL
LIN {X 0,Y 289.137,Z 384.121,A -85,B 0,C 180,E1 -16783.182,E2 -16783.182} C_VEL
LIN {X 0,Y 289.136,Z 383.367,A -85,B 0,C 180,E1 -16785.18,E2 -16785.18} C_VEL
LIN {X 0,Y 289.281,Z 381.815,A -85,B 0,C 180,E1 -16787.138,E2 -16787.138} C_VEL
LIN {X 0,Y 289.499,Z 379.488,A -85,B 0,C 180,E1 -16789.046,E2 -16789.046} C_VEL
LIN {X 0,Y 289.867,Z 376.332,A -85,B 0,C 180,E1 -16790.922,E2 -16790.922} C_VEL
LIN {X 0,Y 290.406,Z 371.807,A -85,B 0,C 180,E1 -16792.997,E2 -16792.997} C_VEL
LIN {X 0,Y 291.054,Z 365.708,A -85,B 0,C 180,E1 -16795.183,E2 -16795.183} C_VEL
LIN {X 0,Y 292.087,Z 357.907,A -85,B 0,C 180,E1 -16797.366,E2 -16797.366} C_VEL
LIN {X 0,Y 293.229,Z 349.412,A -85,B 0,C 180,E1 -16799.275,E2 -16799.275} C_VEL
LIN {X 0,Y 294.347,Z 340.605,A -85,B 0,C 180,E1 -16800.891,E2 -16800.891} C_VEL
LIN {X 0,Y 295.591,Z 330.607,A -85,B 0,C 180,E1 -16802.379,E2 -16802.379} C_VEL
LIN {X 0,Y 296.903,Z 318.75,A -85,B 0,C 180,E1 -16803.783,E2 -16803.783} C_VEL
LIN {X 0,Y 298.066,Z 306.743,A -85,B 0,C 180,E1 -16804.887,E2 -16804.887} C_VEL
LIN {X 0,Y 298.973,Z 293.357,A -85,B 0,C 180,E1 -16805.79,E2 -16805.79} C_VEL
LIN {X 0,Y 299.689,Z 280.298,A -85,B 0,C 180,E1 -16806.386,E2 -16806.386} C_VEL
LIN {X 0,Y 301.903,Z 205.399,A -85,B 0,C 180,E1 -16808.391,E2 -16808.391} C_VEL
LIN {X 0,Y 299.731,Z 193.561,A -85,B 0,C 180,E1 -16808.882,E2 -16808.882} C_VEL
LIN {X 0,Y 292.569,Z 172.909,A -85,B 0,C 180,E1 -16810.027,E2 -16810.027} C_VEL
LIN {X 0,Y 291.432,Z 167.184,A -85,B 0,C 180,E1 -16812.048,E2 -16812.048} C_VEL
LIN {X 0,Y 291.477,Z 167.179,A -85,B 0,C 180,E1 -16816.048,E2 -16816.048} C_VEL
LIN {X 0,Y 291.564,Z 167.169,A -85,B 0,C 180,E1 -16820.286,E2 -16820.286} C_VEL
LIN {X 0,Y 291.683,Z 167.149,A -85,B 0,C 180,E1 -16823.081,E2 -16823.081} C_VEL
LIN {X 0,Y 291.867,Z 167.128,A -85,B 0,C 180,E1 -16828.62,E2 -16828.62} C_VEL
LIN {X 0,Y 291.866,Z 167.128,A -85,B 0,C 180,E1 -16831.38,E2 -16831.38} C_VEL
LIN {X 0,Y 291.682,Z 167.15,A -85,B 0,C 180,E1 -16836.92,E2 -16836.92} C_VEL
LIN {X 0,Y 291.565,Z 167.169,A -85,B 0,C 180,E1 -16839.714,E2 -16839.714} C_VEL
LIN {X 0,Y 291.477,Z 167.179,A -85,B 0,C 180,E1 -16843.952,E2 -16843.952} C_VEL
LIN {X 0,Y 291.399,Z 167.184,A -85,B 0,C 180,E1 -16846.823,E2 -16846.823} C_VEL
LIN {X 0,Y 291.388,Z 167.189,A -85,B 0,C 180,E1 -16849.842,E2 -16849.842} C_VEL
LIN {X 0,Y 291.322,Z 167.194,A -85,B 0,C 180,E1 -16854.212,E2 -16854.212} C_VEL
LIN {X 0,Y 291.324,Z 167.197,A -85,B 0,C 180,E1 -16857.281,E2 -16857.281} C_VEL
LIN {X 0,Y 291.298,Z 167.195,A -85,B 0,C 180,E1 -16860.441,E2 -16860.441} C_VEL
LIN {X 0,Y 291.34,Z 167.193,A -85,B 0,C 180,E1 -16863.699,E2 -16863.699} C_VEL
LIN {X 0,Y 291.355,Z 167.195,A -85,B 0,C 180,E1 -16867.249,E2 -16867.249} C_VEL
LIN {X 0,Y 291.296,Z 167.197,A -85,B 0,C 180,E1 -16870.648,E2 -16870.648} C_VEL
LIN {X 0,Y 291.277,Z 167.197,A -85,B 0,C 180,E1 -16874.404,E2 -16874.404} C_VEL
LIN {X 0,Y 291.29,Z 167.198,A -85,B 0,C 180,E1 -16878.412,E2 -16878.412} C_VEL
LIN {X 0,Y 291.329,Z 167.196,A -85,B 0,C 180,E1 -16881.155,E2 -16881.155} C_VEL
LIN {X 0,Y 291.35,Z 167.191,A -85,B 0,C 180,E1 -16884.625,E2 -16884.625} C_VEL
LIN {X 0,Y 291.361,Z 167.185,A -85,B 0,C 180,E1 -16887.95,E2 -16887.95} C_VEL
LIN {X 0,Y 291.337,Z 167.193,A -85,B 0,C 180,E1 -16891.154,E2 -16891.154} C_VEL
LIN {X 0,Y 291.304,Z 167.194,A -85,B 0,C 180,E1 -16894.977,E2 -16894.977} C_VEL
LIN {X 0,Y 290.63,Z 167.283,A -85,B 0,C 180,E1 -16896.13,E2 -16896.13} C_VEL
LIN {X 0,Y 287.778,Z 167.635,A -85,B 0,C 180,E1 -16898.009,E2 -16898.009} C_VEL
LIN {X 0,Y 285.381,Z 167.93,A -85,B 0,C 180,E1 -16899.535,E2 -16899.535} C_VEL
LIN {X 0,Y 284.377,Z 168.055,A -85,B 0,C 180,E1 -16900.717,E2 -16900.717} C_VEL
LIN {X 0,Y 284.308,Z 168.06,A -85,B 0,C 180,E1 -16901.117,E2 -16901.117} C_VEL
LIN {X 0,Y 284.41,Z 168.057,A -85,B 0,C 180,E1 -16904.517,E2 -16904.517} C_VEL
LIN {X 0,Y 284.453,Z 168.051,A -85,B 0,C 180,E1 -16908.601,E2 -16908.601} C_VEL
LIN {X 0,Y 284.576,Z 168.033,A -85,B 0,C 180,E1 -16911.479,E2 -16911.479} C_VEL
LIN {X 0,Y 284.561,Z 168.034,A -85,B 0,C 180,E1 -16914.331,E2 -16914.331} C_VEL
LIN {X 0,Y 284.831,Z 168.003,A -85,B 0,C 180,E1 -16918.587,E2 -16918.587} C_VEL
LIN {X 0,Y 284.832,Z 168.003,A -85,B 0,C 180,E1 -16921.414,E2 -16921.414} C_VEL
LIN {X 0,Y 284.632,Z 168.023,A -85,B 0,C 180,E1 -16927.092,E2 -16927.092} C_VEL
LIN {X 0,Y 284.508,Z 168.047,A -85,B 0,C 180,E1 -16929.958,E2 -16929.958} C_VEL
LIN {X 0,Y 284.415,Z 168.054,A -85,B 0,C 180,E1 -16934.307,E2 -16934.307} C_VEL
LIN {X 0,Y 284.341,Z 168.062,A -85,B 0,C 180,E1 -16937.254,E2 -16937.254} C_VEL
LIN {X 0,Y 284.32,Z 168.067,A -85,B 0,C 180,E1 -16940.247,E2 -16940.247} C_VEL
LIN {X 0,Y 284.291,Z 168.071,A -85,B 0,C 180,E1 -16943.841,E2 -16943.841} C_VEL
LIN {X 0,Y 284.284,Z 168.074,A -85,B 0,C 180,E1 -16947.13,E2 -16947.13} C_VEL
LIN {X 0,Y 284.272,Z 168.072,A -85,B 0,C 180,E1 -16950.084,E2 -16950.084} C_VEL
LIN {X 0,Y 284.303,Z 168.067,A -85,B 0,C 180,E1 -16952.946,E2 -16952.946} C_VEL
LIN {X 0,Y 284.32,Z 168.066,A -85,B 0,C 180,E1 -16956.389,E2 -16956.389} C_VEL
LIN {X 0,Y 284.281,Z 168.071,A -85,B 0,C 180,E1 -16960,E2 -16960} C_VEL
LIN {X 0,Y 284.233,Z 168.078,A -85,B 0,C 180,E1 -16964.188,E2 -16964.188} C_VEL
LIN {X 0,Y 284.239,Z 168.077,A -85,B 0,C 180,E1 -16968.119,E2 -16968.119} C_VEL
LIN {X 0,Y 284.309,Z 168.069,A -85,B 0,C 180,E1 -16972.282,E2 -16972.282} C_VEL
LIN {X 0,Y 284.308,Z 168.071,A -85,B 0,C 180,E1 -16975.351,E2 -16975.351} C_VEL
LIN {X 0,Y 284.344,Z 168.135,A -85,B 0,C 180,E1 -16977.18,E2 -16977.18} C_VEL
LIN {X 0,Y 286.643,Z 179.471,A -85,B 0,C 180,E1 -16980.954,E2 -16980.954} C_VEL
LIN {X 0,Y 288.275,Z 188,A -85,B 0,C 180,E1 -16983.681,E2 -16983.681} C_VEL
LIN {X 0,Y 289.482,Z 193.093,A -85,B 0,C 180,E1 -16983.934,E2 -16983.934} C_VEL
LIN {X 0,Y 294.741,Z 230.949,A -85,B 0,C 180,E1 -16985.432,E2 -16985.432} C_VEL
LIN {X 0,Y 292.712,Z 297.211,A -85,B 0,C 180,E1 -16987.269,E2 -16987.269} C_VEL
LIN {X 0,Y 291.83,Z 311.106,A -85,B 0,C 180,E1 -16987.943,E2 -16987.943} C_VEL
LIN {X 0,Y 290.812,Z 322.582,A -85,B 0,C 180,E1 -16988.746,E2 -16988.746} C_VEL
LIN {X 0,Y 289.387,Z 335.218,A -85,B 0,C 180,E1 -16989.938,E2 -16989.938} C_VEL
LIN {X 0,Y 287.938,Z 346.535,A -85,B 0,C 180,E1 -16991.316,E2 -16991.316} C_VEL
LIN {X 0,Y 286.701,Z 357.071,A -85,B 0,C 180,E1 -16992.946,E2 -16992.946} C_VEL
LIN {X 0,Y 285.536,Z 366.017,A -85,B 0,C 180,E1 -16994.657,E2 -16994.657} C_VEL
LIN {X 0,Y 284.328,Z 375.011,A -85,B 0,C 180,E1 -16996.783,E2 -16996.783} C_VEL
LIN {X 0,Y 283.417,Z 382.176,A -85,B 0,C 180,E1 -16998.92,E2 -16998.92} C_VEL
LIN {X 0,Y 282.782,Z 388.706,A -85,B 0,C 180,E1 -17001.424,E2 -17001.424} C_VEL
LIN {X 0,Y 282.494,Z 392.969,A -85,B 0,C 180,E1 -17003.572,E2 -17003.572} C_VEL
LIN {X 0,Y 282.348,Z 396.116,A -85,B 0,C 180,E1 -17005.717,E2 -17005.717} C_VEL
LIN {X 0,Y 282.367,Z 397.668,A -85,B 0,C 180,E1 -17007.146,E2 -17007.146} C_VEL
LIN {X 0,Y 282.341,Z 398.742,A -85,B 0,C 180,E1 -17008.573,E2 -17008.573} C_VEL
LIN {X 0,Y 282.357,Z 399.402,A -85,B 0,C 180,E1 -17010,E2 -17010} C_VEL
LIN {X 0,Y 282.331,Z 399.659,A -85,B 0,C 180,E1 -17011.426,E2 -17011.426} C_VEL
LIN {X 0,Y 282.336,Z 399.513,A -85,B 0,C 180,E1 -17012.853,E2 -17012.853} C_VEL
LIN {X 0,Y 282.339,Z 398.255,A -85,B 0,C 180,E1 -17015.32,E2 -17015.32} C_VEL
LIN {X 0,Y 282.577,Z 396.535,A -85,B 0,C 180,E1 -17017.143,E2 -17017.143} C_VEL
LIN {X 0,Y 283.058,Z 393.617,A -85,B 0,C 180,E1 -17019.287,E2 -17019.287} C_VEL
LIN {X 0,Y 283.829,Z 389.665,A -85,B 0,C 180,E1 -17021.425,E2 -17021.425} C_VEL
LIN {X 0,Y 284.915,Z 384.597,A -85,B 0,C 180,E1 -17023.552,E2 -17023.552} C_VEL
LIN {X 0,Y 286.493,Z 378.262,A -85,B 0,C 180,E1 -17025.654,E2 -17025.654} C_VEL
LIN {X 0,Y 287.989,Z 371.634,A -85,B 0,C 180,E1 -17027.443,E2 -17027.443} C_VEL
LIN {X 0,Y 289.577,Z 364.126,A -85,B 0,C 180,E1 -17029.125,E2 -17029.125} C_VEL
LIN {X 0,Y 291.608,Z 354.823,A -85,B 0,C 180,E1 -17030.823,E2 -17030.823} C_VEL
LIN {X 0,Y 294.114,Z 343.231,A -85,B 0,C 180,E1 -17032.477,E2 -17032.477} C_VEL
LIN {X 0,Y 296.113,Z 331.629,A -85,B 0,C 180,E1 -17033.795,E2 -17033.795} C_VEL
LIN {X 0,Y 298.11,Z 318.327,A -85,B 0,C 180,E1 -17034.923,E2 -17034.923} C_VEL
LIN {X 0,Y 299.706,Z 305.447,A -85,B 0,C 180,E1 -17035.71,E2 -17035.71} C_VEL
LIN {X 0,Y 300.776,Z 291.695,A -85,B 0,C 180,E1 -17036.263,E2 -17036.263} C_VEL
LIN {X 0,Y 303.306,Z 232.775,A -85,B 0,C 180,E1 -17037.909,E2 -17037.909} C_VEL
LIN {X 0,Y 300.663,Z 215.195,A -85,B 0,C 180,E1 -17038.866,E2 -17038.866} C_VEL
LIN {X 0,Y 298.787,Z 206.364,A -85,B 0,C 180,E1 -17039.435,E2 -17039.435} C_VEL
LIN {X 0,Y 292.681,Z 193.139,A -85,B 0,C 180,E1 -17040.841,E2 -17040.841} C_VEL
LIN {X 0,Y 288.976,Z 185.587,A -85,B 0,C 180,E1 -17041.779,E2 -17041.779} C_VEL
LIN {X 0,Y 286.946,Z 177.285,A -85,B 0,C 180,E1 -17045.1,E2 -17045.1} C_VEL
LIN {X 0,Y 285,Z 170.577,A -85,B 0,C 180,E1 -17048.059,E2 -17048.059} C_VEL
LIN {X 0,Y 284.265,Z 168.081,A -85,B 0,C 180,E1 -17049.311,E2 -17049.311} C_VEL
LIN {X 0,Y 284.235,Z 168.083,A -85,B 0,C 180,E1 -17052.116,E2 -17052.116} C_VEL
LIN {X 0,Y 284.236,Z 168.082,A -85,B 0,C 180,E1 -17056.185,E2 -17056.185} C_VEL
LIN {X 0,Y 284.281,Z 168.069,A -85,B 0,C 180,E1 -17060.029,E2 -17060.029} C_VEL
LIN {X 0,Y 284.315,Z 168.062,A -85,B 0,C 180,E1 -17063.611,E2 -17063.611} C_VEL
LIN {X 0,Y 284.303,Z 168.064,A -85,B 0,C 180,E1 -17067.189,E2 -17067.189} C_VEL
LIN {X 0,Y 284.309,Z 168.061,A -85,B 0,C 180,E1 -17070.37,E2 -17070.37} C_VEL
LIN {X 0,Y 284.293,Z 168.061,A -85,B 0,C 180,E1 -17073.578,E2 -17073.578} C_VEL
LIN {X 0,Y 284.305,Z 168.062,A -85,B 0,C 180,E1 -17076.701,E2 -17076.701} C_VEL
LIN {X 0,Y 284.33,Z 168.066,A -85,B 0,C 180,E1 -17079.927,E2 -17079.927} C_VEL
LIN {X 0,Y 284.41,Z 168.049,A -85,B 0,C 180,E1 -17084.516,E2 -17084.516} C_VEL
LIN {X 0,Y 284.457,Z 168.044,A -85,B 0,C 180,E1 -17088.6,E2 -17088.6} C_VEL
LIN {X 0,Y 284.602,Z 168.027,A -85,B 0,C 180,E1 -17091.479,E2 -17091.479} C_VEL
LIN {X 0,Y 284.559,Z 168.034,A -85,B 0,C 180,E1 -17094.33,E2 -17094.33} C_VEL
LIN {X 0,Y 284.831,Z 168.002,A -85,B 0,C 180,E1 -17098.586,E2 -17098.586} C_VEL
LIN {X 0,Y 284.831,Z 168.002,A -85,B 0,C 180,E1 -17101.413,E2 -17101.413} C_VEL
LIN {X 0,Y 284.635,Z 168.03,A -85,B 0,C 180,E1 -17107.091,E2 -17107.091} C_VEL
LIN {X 0,Y 284.642,Z 168.194,A -85,B 0,C 180,E1 -17108.888,E2 -17108.888} C_VEL
LIN {X 0,Y 286.395,Z 174.771,A -85,B 0,C 180,E1 -17111.886,E2 -17111.886} C_VEL
LIN {X 0,Y 288.755,Z 178.864,A -85,B 0,C 180,E1 -17112.456,E2 -17112.456} C_VEL
LIN {X 0,Y 295.823,Z 191.901,A -85,B 0,C 180,E1 -17114.079,E2 -17114.079} C_VEL
LIN {X 0,Y 301.68,Z 204.517,A -85,B 0,C 180,E1 -17115.385,E2 -17115.385} C_VEL
LIN {X 0,Y 304.265,Z 211.23,A -85,B 0,C 180,E1 -17115.964,E2 -17115.964} C_VEL
LIN {X 0,Y 300.909,Z 282.507,A -85,B 0,C 180,E1 -17117.96,E2 -17117.96} C_VEL
LIN {X 0,Y 299.78,Z 295.708,A -85,B 0,C 180,E1 -17118.583,E2 -17118.583} C_VEL
LIN {X 0,Y 298.433,Z 308.198,A -85,B 0,C 180,E1 -17119.452,E2 -17119.452} C_VEL
LIN {X 0,Y 296.848,Z 319.234,A -85,B 0,C 180,E1 -17120.47,E2 -17120.47} C_VEL
LIN {X 0,Y 294.995,Z 329.839,A -85,B 0,C 180,E1 -17121.701,E2 -17121.701} C_VEL
LIN {X 0,Y 292.764,Z 340.997,A -85,B 0,C 180,E1 -17123.334,E2 -17123.334} C_VEL
LIN {X 0,Y 290.831,Z 350.086,A -85,B 0,C 180,E1 -17125.017,E2 -17125.017} C_VEL
LIN {X 0,Y 288.953,Z 357.944,A -85,B 0,C 180,E1 -17126.801,E2 -17126.801} C_VEL
LIN {X 0,Y 287.238,Z 365.032,A -85,B 0,C 180,E1 -17128.795,E2 -17128.795} C_VEL
LIN {X 0,Y 285.582,Z 371.57,A -85,B 0,C 180,E1 -17131.117,E2 -17131.117} C_VEL
LIN {X 0,Y 284.162,Z 377.213,A -85,B 0,C 180,E1 -17133.812,E2 -17133.812} C_VEL
LIN {X 0,Y 283.117,Z 381.227,A -85,B 0,C 180,E1 -17136.567,E2 -17136.567} C_VEL
LIN {X 0,Y 282.629,Z 382.978,A -85,B 0,C 180,E1 -17138.437,E2 -17138.437} C_VEL
LIN {X 0,Y 282.309,Z 384.051,A -85,B 0,C 180,E1 -17140.335,E2 -17140.335} C_VEL
LIN {X 0,Y 282.072,Z 384.414,A -85,B 0,C 180,E1 -17142.277,E2 -17142.277} C_VEL
LIN {X 0,Y 282.027,Z 383.975,A -85,B 0,C 180,E1 -17144.246,E2 -17144.246} C_VEL
LIN {X 0,Y 282.093,Z 382.738,A -85,B 0,C 180,E1 -17146.26,E2 -17146.26} C_VEL
LIN {X 0,Y 282.313,Z 380.619,A -85,B 0,C 180,E1 -17148.316,E2 -17148.316} C_VEL
LIN {X 0,Y 282.799,Z 376.405,A -85,B 0,C 180,E1 -17151.026,E2 -17151.026} C_VEL
LIN {X 0,Y 283.426,Z 371.03,A -85,B 0,C 180,E1 -17153.48,E2 -17153.48} C_VEL
LIN {X 0,Y 284.144,Z 364.51,A -85,B 0,C 180,E1 -17155.757,E2 -17155.757} C_VEL
LIN {X 0,Y 285.075,Z 358.041,A -85,B 0,C 180,E1 -17157.575,E2 -17157.575} C_VEL
LIN {X 0,Y 286.27,Z 349.459,A -85,B 0,C 180,E1 -17159.546,E2 -17159.546} C_VEL
LIN {X 0,Y 287.422,Z 340.756,A -85,B 0,C 180,E1 -17161.175,E2 -17161.175} C_VEL
LIN {X 0,Y 288.798,Z 329.932,A -85,B 0,C 180,E1 -17162.805,E2 -17162.805} C_VEL
LIN {X 0,Y 290.053,Z 318.799,A -85,B 0,C 180,E1 -17164.143,E2 -17164.143} C_VEL
LIN {X 0,Y 291.197,Z 307.508,A -85,B 0,C 180,E1 -17165.208,E2 -17165.208} C_VEL
LIN {X 0,Y 292.16,Z 294.118,A -85,B 0,C 180,E1 -17166.146,E2 -17166.146} C_VEL
LIN {X 0,Y 292.895,Z 280.967,A -85,B 0,C 180,E1 -17166.771,E2 -17166.771} C_VEL
LIN {X 0,Y 295.209,Z 206.23,A -85,B 0,C 180,E1 -17168.831,E2 -17168.831} C_VEL
LIN {X 0,Y 293.22,Z 195.561,A -85,B 0,C 180,E1 -17169.286,E2 -17169.286} C_VEL
LIN {X 0,Y 285.361,Z 173.067,A -85,B 0,C 180,E1 -17170.581,E2 -17170.581} C_VEL
LIN {X 0,Y 284.394,Z 168.062,A -85,B 0,C 180,E1 -17172.379,E2 -17172.379} C_VEL
LIN {X 0,Y 284.414,Z 168.058,A -85,B 0,C 180,E1 -17175.694,E2 -17175.694} C_VEL
LIN {X 0,Y 284.51,Z 168.046,A -85,B 0,C 180,E1 -17180.043,E2 -17180.043} C_VEL
LIN {X 0,Y 284.639,Z 168.027,A -85,B 0,C 180,E1 -17182.909,E2 -17182.909} C_VEL
LIN {X 0,Y 284.834,Z 168.005,A -85,B 0,C 180,E1 -17188.586,E2 -17188.586} C_VEL
LIN {X 0,Y 284.833,Z 168.004,A -85,B 0,C 180,E1 -17191.414,E2 -17191.414} C_VEL
LIN {X 0,Y 284.638,Z 168.028,A -85,B 0,C 180,E1 -17197.092,E2 -17197.092} C_VEL
LIN {X 0,Y 284.51,Z 168.048,A -85,B 0,C 180,E1 -17199.957,E2 -17199.957} C_VEL
LIN {X 0,Y 284.414,Z 168.056,A -85,B 0,C 180,E1 -17204.306,E2 -17204.306} C_VEL
LIN {X 0,Y 284.313,Z 168.067,A -85,B 0,C 180,E1 -17208.745,E2 -17208.745} C_VEL
LIN {X 0,Y 284.294,Z 168.073,A -85,B 0,C 180,E1 -17211.766,E2 -17211.766} C_VEL
LIN {X 0,Y 284.279,Z 168.071,A -85,B 0,C 180,E1 -17214.852,E2 -17214.852} C_VEL
LIN {X 0,Y 284.256,Z 168.075,A -85,B 0,C 180,E1 -17218.019,E2 -17218.019} C_VEL
LIN {X 0,Y 284.274,Z 168.074,A -85,B 0,C 180,E1 -17221.277,E2 -17221.277} C_VEL
LIN {X 0,Y 284.333,Z 168.069,A -85,B 0,C 180,E1 -17225.347,E2 -17225.347} C_VEL
LIN {X 0,Y 284.294,Z 168.069,A -85,B 0,C 180,E1 -17228.172,E2 -17228.172} C_VEL
LIN {X 0,Y 284.232,Z 168.074,A -85,B 0,C 180,E1 -17232.117,E2 -17232.117} C_VEL
LIN {X 0,Y 284.233,Z 168.075,A -85,B 0,C 180,E1 -17236.186,E2 -17236.186} C_VEL
LIN {X 0,Y 284.279,Z 168.071,A -85,B 0,C 180,E1 -17240.03,E2 -17240.03} C_VEL
LIN {X 0,Y 284.316,Z 168.065,A -85,B 0,C 180,E1 -17243.612,E2 -17243.612} C_VEL
LIN {X 0,Y 284.302,Z 168.065,A -85,B 0,C 180,E1 -17247.191,E2 -17247.191} C_VEL
LIN {X 0,Y 284.332,Z 168.065,A -85,B 0,C 180,E1 -17250.374,E2 -17250.374} C_VEL
LIN {X 0,Y 284.292,Z 168.07,A -85,B 0,C 180,E1 -17253.579,E2 -17253.579} C_VEL
LIN {X 0,Y 284.303,Z 168.071,A -85,B 0,C 180,E1 -17256.702,E2 -17256.702} C_VEL
LIN {X 0,Y 284.308,Z 168.06,A -85,B 0,C 180,E1 -17261.117,E2 -17261.117} C_VEL
LIN {X 0,Y 283.679,Z 168.144,A -85,B 0,C 180,E1 -17262.301,E2 -17262.301} C_VEL
LIN {X 0,Y 280.863,Z 168.496,A -85,B 0,C 180,E1 -17264.23,E2 -17264.23} C_VEL
LIN {X 0,Y 278.46,Z 168.795,A -85,B 0,C 180,E1 -17265.797,E2 -17265.797} C_VEL
LIN {X 0,Y 277.438,Z 168.924,A -85,B 0,C 180,E1 -17267.01,E2 -17267.01} C_VEL
LIN {X 0,Y 277.36,Z 168.932,A -85,B 0,C 180,E1 -17267.421,E2 -17267.421} C_VEL
LIN {X 0,Y 277.547,Z 168.908,A -85,B 0,C 180,E1 -17271.262,E2 -17271.262} C_VEL
LIN {X 0,Y 277.531,Z 168.91,A -85,B 0,C 180,E1 -17274.187,E2 -17274.187} C_VEL
LIN {X 0,Y 277.798,Z 168.879,A -85,B 0,C 180,E1 -17278.551,E2 -17278.551} C_VEL
LIN {X 0,Y 277.799,Z 168.879,A -85,B 0,C 180,E1 -17281.45,E2 -17281.45} C_VEL
LIN {X 0,Y 277.588,Z 168.9,A -85,B 0,C 180,E1 -17287.273,E2 -17287.273} C_VEL
LIN {X 0,Y 277.449,Z 168.924,A -85,B 0,C 180,E1 -17290.214,E2 -17290.214} C_VEL
LIN {X 0,Y 277.368,Z 168.931,A -85,B 0,C 180,E1 -17294.678,E2 -17294.678} C_VEL
LIN {X 0,Y 277.272,Z 168.945,A -85,B 0,C 180,E1 -17299.24,E2 -17299.24} C_VEL
LIN {X 0,Y 277.253,Z 168.947,A -85,B 0,C 180,E1 -17303.928,E2 -17303.928} C_VEL
LIN {X 0,Y 277.233,Z 168.955,A -85,B 0,C 180,E1 -17307.469,E2 -17307.469} C_VEL
LIN {X 0,Y 277.227,Z 168.949,A -85,B 0,C 180,E1 -17310.466,E2 -17310.466} C_VEL
LIN {X 0,Y 277.245,Z 168.944,A -85,B 0,C 180,E1 -17313.897,E2 -17313.897} C_VEL
LIN {X 0,Y 277.254,Z 168.95,A -85,B 0,C 180,E1 -17317.472,E2 -17317.472} C_VEL
LIN {X 0,Y 277.183,Z 168.96,A -85,B 0,C 180,E1 -17321.242,E2 -17321.242} C_VEL
LIN {X 0,Y 277.173,Z 168.96,A -85,B 0,C 180,E1 -17325.233,E2 -17325.233} C_VEL
LIN {X 0,Y 277.184,Z 168.959,A -85,B 0,C 180,E1 -17328.759,E2 -17328.759} C_VEL
LIN {X 0,Y 277.255,Z 168.949,A -85,B 0,C 180,E1 -17332.529,E2 -17332.529} C_VEL
LIN {X 0,Y 277.254,Z 168.949,A -85,B 0,C 180,E1 -17336.106,E2 -17336.106} C_VEL
LIN {X 0,Y 277.291,Z 169.132,A -85,B 0,C 180,E1 -17336.836,E2 -17336.836} C_VEL
LIN {X 0,Y 279.595,Z 180.297,A -85,B 0,C 180,E1 -17340.65,E2 -17340.65} C_VEL
LIN {X 0,Y 281.051,Z 187.887,A -85,B 0,C 180,E1 -17343.138,E2 -17343.138} C_VEL
LIN {X 0,Y 282.881,Z 194.349,A -85,B 0,C 180,E1 -17343.482,E2 -17343.482} C_VEL
LIN {X 0,Y 288.012,Z 231.632,A -85,B 0,C 180,E1 -17344.998,E2 -17344.998} C_VEL
LIN {X 0,Y 285.943,Z 296.634,A -85,B 0,C 180,E1 -17346.843,E2 -17346.843} C_VEL
LIN {X 0,Y 285.03,Z 310.632,A -85,B 0,C 180,E1 -17347.531,E2 -17347.531} C_VEL
LIN {X 0,Y 283.953,Z 322.713,A -85,B 0,C 180,E1 -17348.398,E2 -17348.398} C_VEL
LIN {X 0,Y 282.487,Z 335.27,A -85,B 0,C 180,E1 -17349.616,E2 -17349.616} C_VEL
LIN {X 0,Y 280.999,Z 346.544,A -85,B 0,C 180,E1 -17351.026,E2 -17351.026} C_VEL
LIN {X 0,Y 279.699,Z 357.141,A -85,B 0,C 180,E1 -17352.715,E2 -17352.715} C_VEL
LIN {X 0,Y 278.388,Z 366.785,A -85,B 0,C 180,E1 -17354.629,E2 -17354.629} C_VEL
LIN {X 0,Y 277.383,Z 374.242,A -85,B 0,C 180,E1 -17356.446,E2 -17356.446} C_VEL
LIN {X 0,Y 276.407,Z 381.55,A -85,B 0,C 180,E1 -17358.635,E2 -17358.635} C_VEL
LIN {X 0,Y 275.893,Z 386.472,A -85,B 0,C 180,E1 -17360.469,E2 -17360.469} C_VEL
LIN {X 0,Y 275.505,Z 391.22,A -85,B 0,C 180,E1 -17362.672,E2 -17362.672} C_VEL
LIN {X 0,Y 275.329,Z 394.357,A -85,B 0,C 180,E1 -17364.573,E2 -17364.573} C_VEL
LIN {X 0,Y 275.276,Z 397.325,A -85,B 0,C 180,E1 -17367.073,E2 -17367.073} C_VEL
LIN {X 0,Y 275.266,Z 398.464,A -85,B 0,C 180,E1 -17368.537,E2 -17368.537} C_VEL
LIN {X 0,Y 275.279,Z 399.156,A -85,B 0,C 180,E1 -17370,E2 -17370} C_VEL
LIN {X 0,Y 275.256,Z 399.445,A -85,B 0,C 180,E1 -17371.463,E2 -17371.463} C_VEL
LIN {X 0,Y 275.245,Z 399.335,A -85,B 0,C 180,E1 -17372.927,E2 -17372.927} C_VEL
LIN {X 0,Y 275.24,Z 398.307,A -85,B 0,C 180,E1 -17375.228,E2 -17375.228} C_VEL
LIN {X 0,Y 275.512,Z 396.474,A -85,B 0,C 180,E1 -17377.327,E2 -17377.327} C_VEL
LIN {X 0,Y 276.018,Z 393.632,A -85,B 0,C 180,E1 -17379.526,E2 -17379.526} C_VEL
LIN {X 0,Y 276.863,Z 389.767,A -85,B 0,C 180,E1 -17381.716,E2 -17381.716} C_VEL
LIN {X 0,Y 277.997,Z 384.785,A -85,B 0,C 180,E1 -17383.896,E2 -17383.896} C_VEL
LIN {X 0,Y 279.68,Z 378.534,A -85,B 0,C 180,E1 -17386.046,E2 -17386.046} C_VEL
LIN {X 0,Y 281.169,Z 372.201,A -85,B 0,C 180,E1 -17387.825,E2 -17387.825} C_VEL
LIN {X 0,Y 283.308,Z 362.932,A -85,B 0,C 180,E1 -17389.943,E2 -17389.943} C_VEL
LIN {X 0,Y 285.779,Z 352.32,A -85,B 0,C 180,E1 -17391.836,E2 -17391.836} C_VEL
LIN {X 0,Y 288.126,Z 341.606,A -85,B 0,C 180,E1 -17393.351,E2 -17393.351} C_VEL
LIN {X 0,Y 290.293,Z 329.579,A -85,B 0,C 180,E1 -17394.684,E2 -17394.684} C_VEL
LIN {X 0,Y 292.266,Z 316.92,A -85,B 0,C 180,E1 -17395.743,E2 -17395.743} C_VEL
LIN {X 0,Y 293.842,Z 304.25,A -85,B 0,C 180,E1 -17396.5,E2 -17396.5} C_VEL
LIN {X 0,Y 294.901,Z 290.666,A -85,B 0,C 180,E1 -17397.041,E2 -17397.041} C_VEL
LIN {X 0,Y 297.482,Z 234.397,A -85,B 0,C 180,E1 -17398.636,E2 -17398.636} C_VEL
LIN {X 0,Y 295.376,Z 219.157,A -85,B 0,C 180,E1 -17399.477,E2 -17399.477} C_VEL
LIN {X 0,Y 293.54,Z 209.716,A -85,B 0,C 180,E1 -17400.098,E2 -17400.098} C_VEL
LIN {X 0,Y 286.622,Z 194.655,A -85,B 0,C 180,E1 -17401.771,E2 -17401.771} C_VEL
LIN {X 0,Y 283.067,Z 188.27,A -85,B 0,C 180,E1 -17402.646,E2 -17402.646} C_VEL
LIN {X 0,Y 281.78,Z 185.402,A -85,B 0,C 180,E1 -17403.013,E2 -17403.013} C_VEL
LIN {X 0,Y 279.708,Z 177.271,A -85,B 0,C 180,E1 -17406.482,E2 -17406.482} C_VEL
LIN {X 0,Y 277.201,Z 168.958,A -85,B 0,C 180,E1 -17410.525,E2 -17410.525} C_VEL
LIN {X 0,Y 277.172,Z 168.959,A -85,B 0,C 180,E1 -17414.767,E2 -17414.767} C_VEL
LIN {X 0,Y 277.181,Z 168.959,A -85,B 0,C 180,E1 -17418.758,E2 -17418.758} C_VEL
LIN {X 0,Y 277.248,Z 168.947,A -85,B 0,C 180,E1 -17422.527,E2 -17422.527} C_VEL
LIN {X 0,Y 277.243,Z 168.944,A -85,B 0,C 180,E1 -17426.103,E2 -17426.103} C_VEL
LIN {X 0,Y 277.225,Z 168.944,A -85,B 0,C 180,E1 -17429.533,E2 -17429.533} C_VEL
LIN {X 0,Y 277.25,Z 168.942,A -85,B 0,C 180,E1 -17432.852,E2 -17432.852} C_VEL
LIN {X 0,Y 277.256,Z 168.947,A -85,B 0,C 180,E1 -17436.072,E2 -17436.072} C_VEL
LIN {X 0,Y 277.27,Z 168.937,A -85,B 0,C 180,E1 -17440.76,E2 -17440.76} C_VEL
LIN {X 0,Y 277.366,Z 168.927,A -85,B 0,C 180,E1 -17445.322,E2 -17445.322} C_VEL
LIN {X 0,Y 277.449,Z 168.924,A -85,B 0,C 180,E1 -17449.786,E2 -17449.786} C_VEL
LIN {X 0,Y 277.594,Z 168.903,A -85,B 0,C 180,E1 -17452.727,E2 -17452.727} C_VEL
LIN {X 0,Y 277.798,Z 168.877,A -85,B 0,C 180,E1 -17458.55,E2 -17458.55} C_VEL
LIN {X 0,Y 277.798,Z 168.878,A -85,B 0,C 180,E1 -17461.449,E2 -17461.449} C_VEL
LIN {X 0,Y 277.58,Z 168.907,A -85,B 0,C 180,E1 -17467.455,E2 -17467.455} C_VEL
LIN {X 0,Y 278.251,Z 171.168,A -85,B 0,C 180,E1 -17468.716,E2 -17468.716} C_VEL
LIN {X 0,Y 279.195,Z 175.029,A -85,B 0,C 180,E1 -17470.561,E2 -17470.561} C_VEL
LIN {X 0,Y 281.765,Z 179.349,A -85,B 0,C 180,E1 -17471.236,E2 -17471.236} C_VEL
LIN {X 0,Y 288.86,Z 191.894,A -85,B 0,C 180,E1 -17472.981,E2 -17472.981} C_VEL
LIN {X 0,Y 295.199,Z 205.03,A -85,B 0,C 180,E1 -17474.462,E2 -17474.462} C_VEL
LIN {X 0,Y 298.339,Z 212.713,A -85,B 0,C 180,E1 -17475.205,E2 -17475.205} C_VEL
LIN {X 0,Y 294.932,Z 283.16,A -85,B 0,C 180,E1 -17477.231,E2 -17477.231} C_VEL
LIN {X 0,Y 293.713,Z 296.711,A -85,B 0,C 180,E1 -17477.892,E2 -17477.892} C_VEL
LIN {X 0,Y 292.328,Z 308.75,A -85,B 0,C 180,E1 -17478.756,E2 -17478.756} C_VEL
LIN {X 0,Y 290.697,Z 319.624,A -85,B 0,C 180,E1 -17479.783,E2 -17479.783} C_VEL
LIN {X 0,Y 288.748,Z 330.188,A -85,B 0,C 180,E1 -17481.039,E2 -17481.039} C_VEL
LIN {X 0,Y 286.563,Z 340.66,A -85,B 0,C 180,E1 -17482.602,E2 -17482.602} C_VEL
LIN {X 0,Y 284.375,Z 350.223,A -85,B 0,C 180,E1 -17484.393,E2 -17484.393} C_VEL
LIN {X 0,Y 282.283,Z 358.524,A -85,B 0,C 180,E1 -17486.328,E2 -17486.328} C_VEL
LIN {X 0,Y 280.257,Z 366.394,A -85,B 0,C 180,E1 -17488.637,E2 -17488.637} C_VEL
LIN {X 0,Y 278.596,Z 372.51,A -85,B 0,C 180,E1 -17490.943,E2 -17490.943} C_VEL
LIN {X 0,Y 277.344,Z 377.188,A -85,B 0,C 180,E1 -17493.257,E2 -17493.257} C_VEL
LIN {X 0,Y 276.262,Z 380.934,A -85,B 0,C 180,E1 -17495.81,E2 -17495.81} C_VEL
LIN {X 0,Y 275.682,Z 382.915,A -85,B 0,C 180,E1 -17497.789,E2 -17497.789} C_VEL
LIN {X 0,Y 275.259,Z 384.227,A -85,B 0,C 180,E1 -17500.008,E2 -17500.008} C_VEL
LIN {X 0,Y 274.984,Z 384.616,A -85,B 0,C 180,E1 -17502.169,E2 -17502.169} C_VEL
LIN {X 0,Y 274.927,Z 384.109,A -85,B 0,C 180,E1 -17504.295,E2 -17504.295} C_VEL
LIN {X 0,Y 274.999,Z 382.78,A -85,B 0,C 180,E1 -17506.369,E2 -17506.369} C_VEL
LIN {X 0,Y 275.22,Z 380.666,A -85,B 0,C 180,E1 -17508.401,E2 -17508.401} C_VEL
LIN {X 0,Y 275.54,Z 377.785,A -85,B 0,C 180,E1 -17510.384,E2 -17510.384} C_VEL
LIN {X 0,Y 276.149,Z 373.008,A -85,B 0,C 180,E1 -17512.813,E2 -17512.813} C_VEL
LIN {X 0,Y 276.885,Z 366.707,A -85,B 0,C 180,E1 -17515.253,E2 -17515.253} C_VEL
LIN {X 0,Y 277.988,Z 358.736,A -85,B 0,C 180,E1 -17517.639,E2 -17517.639} C_VEL
LIN {X 0,Y 279.271,Z 349.683,A -85,B 0,C 180,E1 -17519.781,E2 -17519.781} C_VEL
LIN {X 0,Y 280.598,Z 340.191,A -85,B 0,C 180,E1 -17521.584,E2 -17521.584} C_VEL
LIN {X 0,Y 281.909,Z 330.026,A -85,B 0,C 180,E1 -17523.138,E2 -17523.138} C_VEL
LIN {X 0,Y 283.162,Z 319.334,A -85,B 0,C 180,E1 -17524.454,E2 -17524.454} C_VEL
LIN {X 0,Y 284.351,Z 307.72,A -85,B 0,C 180,E1 -17525.581,E2 -17525.581} C_VEL
LIN {X 0,Y 285.313,Z 295.138,A -85,B 0,C 180,E1 -17526.493,E2 -17526.493} C_VEL
LIN {X 0,Y 286.089,Z 281.545,A -85,B 0,C 180,E1 -17527.167,E2 -17527.167} C_VEL
LIN {X 0,Y 288.541,Z 207.107,A -85,B 0,C 180,E1 -17529.272,E2 -17529.272} C_VEL
LIN {X 0,Y 286.699,Z 197.615,A -85,B 0,C 180,E1 -17529.695,E2 -17529.695} C_VEL
LIN {X 0,Y 278.205,Z 173.357,A -85,B 0,C 180,E1 -17531.116,E2 -17531.116} C_VEL
LIN {X 0,Y 277.35,Z 168.939,A -85,B 0,C 180,E1 -17532.773,E2 -17532.773} C_VEL
LIN {X 0,Y 277.371,Z 168.936,A -85,B 0,C 180,E1 -17536.819,E2 -17536.819} C_VEL
LIN {X 0,Y 277.567,Z 168.907,A -85,B 0,C 180,E1 -17541.262,E2 -17541.262} C_VEL
LIN {X 0,Y 277.534,Z 168.916,A -85,B 0,C 180,E1 -17544.187,E2 -17544.187} C_VEL
LIN {X 0,Y 277.801,Z 168.881,A -85,B 0,C 180,E1 -17548.551,E2 -17548.551} C_VEL
LIN {X 0,Y 277.799,Z 168.881,A -85,B 0,C 180,E1 -17551.45,E2 -17551.45} C_VEL
LIN {X 0,Y 277.597,Z 168.905,A -85,B 0,C 180,E1 -17557.273,E2 -17557.273} C_VEL
LIN {X 0,Y 277.45,Z 168.925,A -85,B 0,C 180,E1 -17560.213,E2 -17560.213} C_VEL
LIN {X 0,Y 277.367,Z 168.933,A -85,B 0,C 180,E1 -17564.678,E2 -17564.678} C_VEL
LIN {X 0,Y 277.273,Z 168.946,A -85,B 0,C 180,E1 -17569.239,E2 -17569.239} C_VEL
LIN {X 0,Y 277.251,Z 168.948,A -85,B 0,C 180,E1 -17573.927,E2 -17573.927} C_VEL
LIN {X 0,Y 277.231,Z 168.954,A -85,B 0,C 180,E1 -17577.469,E2 -17577.469} C_VEL
LIN {X 0,Y 277.224,Z 168.948,A -85,B 0,C 180,E1 -17580.466,E2 -17580.466} C_VEL
LIN {X 0,Y 277.242,Z 168.947,A -85,B 0,C 180,E1 -17583.896,E2 -17583.896} C_VEL
LIN {X 0,Y 277.251,Z 168.95,A -85,B 0,C 180,E1 -17587.472,E2 -17587.472} C_VEL
LIN {X 0,Y 277.179,Z 168.956,A -85,B 0,C 180,E1 -17591.242,E2 -17591.242} C_VEL
LIN {X 0,Y 277.169,Z 168.958,A -85,B 0,C 180,E1 -17595.233,E2 -17595.233} C_VEL
LIN {X 0,Y 277.18,Z 168.958,A -85,B 0,C 180,E1 -17598.759,E2 -17598.759} C_VEL
LIN {X 0,Y 277.25,Z 168.948,A -85,B 0,C 180,E1 -17602.529,E2 -17602.529} C_VEL
LIN {X 0,Y 277.241,Z 168.942,A -85,B 0,C 180,E1 -17606.104,E2 -17606.104} C_VEL
LIN {X 0,Y 277.258,Z 168.943,A -85,B 0,C 180,E1 -17609.539,E2 -17609.539} C_VEL
LIN {X 0,Y 277.284,Z 168.946,A -85,B 0,C 180,E1 -17612.857,E2 -17612.857} C_VEL
LIN {X 0,Y 277.251,Z 168.948,A -85,B 0,C 180,E1 -17616.073,E2 -17616.073} C_VEL
LIN {X 0,Y 277.272,Z 168.939,A -85,B 0,C 180,E1 -17620.762,E2 -17620.762} C_VEL
LIN {X 0,Y 277.367,Z 168.93,A -85,B 0,C 180,E1 -17625.323,E2 -17625.323} C_VEL
LIN {X 0,Y 277.36,Z 168.932,A -85,B 0,C 180,E1 -17627.421,E2 -17627.421} C_VEL
LIN {X 0,Y 276.721,Z 169.015,A -85,B 0,C 180,E1 -17628.634,E2 -17628.634} C_VEL
LIN {X 0,Y 273.932,Z 169.36,A -85,B 0,C 180,E1 -17630.613,E2 -17630.613} C_VEL
LIN {X 0,Y 271.569,Z 169.655,A -85,B 0,C 180,E1 -17632.221,E2 -17632.221} C_VEL
LIN {X 0,Y 270.571,Z 169.775,A -85,B 0,C 180,E1 -17633.465,E2 -17633.465} C_VEL
LIN {X 0,Y 270.498,Z 169.785,A -85,B 0,C 180,E1 -17633.887,E2 -17633.887} C_VEL
LIN {X 0,Y 270.764,Z 169.755,A -85,B 0,C 180,E1 -17638.513,E2 -17638.513} C_VEL
LIN {X 0,Y 270.764,Z 169.755,A -85,B 0,C 180,E1 -17641.488,E2 -17641.488} C_VEL
LIN {X 0,Y 270.549,Z 169.777,A -85,B 0,C 180,E1 -17647.464,E2 -17647.464} C_VEL
LIN {X 0,Y 270.381,Z 169.803,A -85,B 0,C 180,E1 -17650.484,E2 -17650.484} C_VEL
LIN {X 0,Y 270.336,Z 169.808,A -85,B 0,C 180,E1 -17655.069,E2 -17655.069} C_VEL
LIN {X 0,Y 270.216,Z 169.827,A -85,B 0,C 180,E1 -17659.763,E2 -17659.763} C_VEL
LIN {X 0,Y 270.18,Z 169.826,A -85,B 0,C 180,E1 -17664.436,E2 -17664.436} C_VEL
LIN {X 0,Y 270.183,Z 169.83,A -85,B 0,C 180,E1 -17667.919,E2 -17667.919} C_VEL
LIN {X 0,Y 270.168,Z 169.83,A -85,B 0,C 180,E1 -17671.351,E2 -17671.351} C_VEL
LIN {X 0,Y 270.197,Z 169.823,A -85,B 0,C 180,E1 -17674.907,E2 -17674.907} C_VEL
LIN {X 0,Y 270.198,Z 169.827,A -85,B 0,C 180,E1 -17678.711,E2 -17678.711} C_VEL
LIN {X 0,Y 270.147,Z 169.836,A -85,B 0,C 180,E1 -17683.245,E2 -17683.245} C_VEL
LIN {X 0,Y 270.151,Z 169.833,A -85,B 0,C 180,E1 -17687.438,E2 -17687.438} C_VEL
LIN {X 0,Y 270.209,Z 169.827,A -85,B 0,C 180,E1 -17691.375,E2 -17691.375} C_VEL
LIN {X 0,Y 270.201,Z 169.829,A -85,B 0,C 180,E1 -17695.095,E2 -17695.095} C_VEL
LIN {X 0,Y 270.219,Z 169.886,A -85,B 0,C 180,E1 -17696.39,E2 -17696.39} C_VEL
LIN {X 0,Y 272.492,Z 180.809,A -85,B 0,C 180,E1 -17700.232,E2 -17700.232} C_VEL
LIN {X 0,Y 273.862,Z 187.804,A -85,B 0,C 180,E1 -17702.559,E2 -17702.559} C_VEL
LIN {X 0,Y 276.327,Z 195.889,A -85,B 0,C 180,E1 -17703.019,E2 -17703.019} C_VEL
LIN {X 0,Y 281.305,Z 232.515,A -85,B 0,C 180,E1 -17704.553,E2 -17704.553} C_VEL
LIN {X 0,Y 279.205,Z 296.065,A -85,B 0,C 180,E1 -17706.398,E2 -17706.398} C_VEL
LIN {X 0,Y 278.26,Z 310.163,A -85,B 0,C 180,E1 -17707.101,E2 -17707.101} C_VEL
LIN {X 0,Y 277.104,Z 322.832,A -85,B 0,C 180,E1 -17708.032,E2 -17708.032} C_VEL
LIN {X 0,Y 275.582,Z 335.319,A -85,B 0,C 180,E1 -17709.277,E2 -17709.277} C_VEL
LIN {X 0,Y 274.069,Z 346.554,A -85,B 0,C 180,E1 -17710.722,E2 -17710.722} C_VEL
LIN {X 0,Y 272.688,Z 357.258,A -85,B 0,C 180,E1 -17712.48,E2 -17712.48} C_VEL
LIN {X 0,Y 271.521,Z 365.899,A -85,B 0,C 180,E1 -17714.23,E2 -17714.23} C_VEL
LIN {X 0,Y 270.228,Z 374.851,A -85,B 0,C 180,E1 -17716.463,E2 -17716.463} C_VEL
LIN {X 0,Y 269.282,Z 381.966,A -85,B 0,C 180,E1 -17718.712,E2 -17718.712} C_VEL
LIN {X 0,Y 268.68,Z 387.639,A -85,B 0,C 180,E1 -17720.97,E2 -17720.97} C_VEL
LIN {X 0,Y 268.333,Z 392.061,A -85,B 0,C 180,E1 -17723.231,E2 -17723.231} C_VEL
LIN {X 0,Y 268.179,Z 395.356,A -85,B 0,C 180,E1 -17725.491,E2 -17725.491} C_VEL
LIN {X 0,Y 268.187,Z 396.98,A -85,B 0,C 180,E1 -17726.995,E2 -17726.995} C_VEL
LIN {X 0,Y 268.192,Z 398.178,A -85,B 0,C 180,E1 -17728.498,E2 -17728.498} C_VEL
LIN {X 0,Y 268.202,Z 398.91,A -85,B 0,C 180,E1 -17730,E2 -17730} C_VEL
LIN {X 0,Y 268.182,Z 399.23,A -85,B 0,C 180,E1 -17731.501,E2 -17731.501} C_VEL
LIN {X 0,Y 268.156,Z 399.153,A -85,B 0,C 180,E1 -17733.004,E2 -17733.004} C_VEL
LIN {X 0,Y 268.165,Z 398.296,A -85,B 0,C 180,E1 -17735.187,E2 -17735.187} C_VEL
LIN {X 0,Y 268.453,Z 396.436,A -85,B 0,C 180,E1 -17737.521,E2 -17737.521} C_VEL
LIN {X 0,Y 268.997,Z 393.666,A -85,B 0,C 180,E1 -17739.777,E2 -17739.777} C_VEL
LIN {X 0,Y 269.887,Z 389.877,A -85,B 0,C 180,E1 -17742.024,E2 -17742.024} C_VEL
LIN {X 0,Y 271.098,Z 384.973,A -85,B 0,C 180,E1 -17744.257,E2 -17744.257} C_VEL
LIN {X 0,Y 273.223,Z 377.671,A -85,B 0,C 180,E1 -17746.82,E2 -17746.82} C_VEL
LIN {X 0,Y 275.156,Z 369.495,A -85,B 0,C 180,E1 -17749.081,E2 -17749.081} C_VEL
LIN {X 0,Y 277.172,Z 361.777,A -85,B 0,C 180,E1 -17750.792,E2 -17750.792} C_VEL
LIN {X 0,Y 279.525,Z 352.065,A -85,B 0,C 180,E1 -17752.545,E2 -17752.545} C_VEL
LIN {X 0,Y 281.964,Z 341.338,A -85,B 0,C 180,E1 -17754.088,E2 -17754.088} C_VEL
LIN {X 0,Y 284.242,Z 329.286,A -85,B 0,C 180,E1 -17755.442,E2 -17755.442} C_VEL
LIN {X 0,Y 286.316,Z 316.602,A -85,B 0,C 180,E1 -17756.515,E2 -17756.515} C_VEL
LIN {X 0,Y 287.936,Z 303.89,A -85,B 0,C 180,E1 -17757.284,E2 -17757.284} C_VEL
LIN {X 0,Y 289.032,Z 290.325,A -85,B 0,C 180,E1 -17757.832,E2 -17757.832} C_VEL
LIN {X 0,Y 291.712,Z 235.162,A -85,B 0,C 180,E1 -17759.441,E2 -17759.441} C_VEL
LIN {X 0,Y 289.592,Z 219.886,A -85,B 0,C 180,E1 -17760.33,E2 -17760.33} C_VEL
LIN {X 0,Y 288.187,Z 212.868,A -85,B 0,C 180,E1 -17760.816,E2 -17760.816} C_VEL
LIN {X 0,Y 281.994,Z 199.042,A -85,B 0,C 180,E1 -17762.405,E2 -17762.405} C_VEL
LIN {X 0,Y 276.583,Z 189.103,A -85,B 0,C 180,E1 -17763.824,E2 -17763.824} C_VEL
LIN {X 0,Y 274.505,Z 185.109,A -85,B 0,C 180,E1 -17764.419,E2 -17764.419} C_VEL
LIN {X 0,Y 273.01,Z 179.252,A -85,B 0,C 180,E1 -17767.058,E2 -17767.058} C_VEL
LIN {X 0,Y 271.001,Z 172.524,A -85,B 0,C 180,E1 -17770.415,E2 -17770.415} C_VEL
LIN {X 0,Y 270.138,Z 169.84,A -85,B 0,C 180,E1 -17771.933,E2 -17771.933} C_VEL
LIN {X 0,Y 270.127,Z 169.836,A -85,B 0,C 180,E1 -17775.374,E2 -17775.374} C_VEL
LIN {X 0,Y 270.146,Z 169.833,A -85,B 0,C 180,E1 -17779.428,E2 -17779.428} C_VEL
LIN {X 0,Y 270.204,Z 169.819,A -85,B 0,C 180,E1 -17783.256,E2 -17783.256} C_VEL
LIN {X 0,Y 270.198,Z 169.819,A -85,B 0,C 180,E1 -17786.891,E2 -17786.891} C_VEL
LIN {X 0,Y 270.155,Z 169.823,A -85,B 0,C 180,E1 -17790.377,E2 -17790.377} C_VEL
LIN {X 0,Y 270.176,Z 169.82,A -85,B 0,C 180,E1 -17793.754,E2 -17793.754} C_VEL
LIN {X 0,Y 270.178,Z 169.82,A -85,B 0,C 180,E1 -17797.033,E2 -17797.033} C_VEL
LIN {X 0,Y 270.214,Z 169.82,A -85,B 0,C 180,E1 -17800.237,E2 -17800.237} C_VEL
LIN {X 0,Y 270.333,Z 169.801,A -85,B 0,C 180,E1 -17804.931,E2 -17804.931} C_VEL
LIN {X 0,Y 270.382,Z 169.803,A -85,B 0,C 180,E1 -17809.516,E2 -17809.516} C_VEL
LIN {X 0,Y 270.556,Z 169.778,A -85,B 0,C 180,E1 -17812.537,E2 -17812.537} C_VEL
LIN {X 0,Y 270.763,Z 169.753,A -85,B 0,C 180,E1 -17818.512,E2 -17818.512} C_VEL
LIN {X 0,Y 270.763,Z 169.755,A -85,B 0,C 180,E1 -17821.487,E2 -17821.487} C_VEL
LIN {X 0,Y 270.503,Z 169.921,A -85,B 0,C 180,E1 -17826.245,E2 -17826.245} C_VEL
LIN {X 0,Y 272.13,Z 175.381,A -85,B 0,C 180,E1 -17829.148,E2 -17829.148} C_VEL
LIN {X 0,Y 274.455,Z 179.363,A -85,B 0,C 180,E1 -17829.813,E2 -17829.813} C_VEL
LIN {X 0,Y 280.528,Z 189.516,A -85,B 0,C 180,E1 -17831.424,E2 -17831.424} C_VEL
LIN {X 0,Y 287.329,Z 202.551,A -85,B 0,C 180,E1 -17833.136,E2 -17833.136} C_VEL
LIN {X 0,Y 292.59,Z 214.878,A -85,B 0,C 180,E1 -17834.426,E2 -17834.426} C_VEL
LIN {X 0,Y 289.101,Z 283.04,A -85,B 0,C 180,E1 -17836.438,E2 -17836.438} C_VEL
LIN {X 0,Y 287.798,Z 296.795,A -85,B 0,C 180,E1 -17837.118,E2 -17837.118} C_VEL
LIN {X 0,Y 286.241,Z 309.464,A -85,B 0,C 180,E1 -17838.047,E2 -17838.047} C_VEL
LIN {X 0,Y 284.411,Z 321.014,A -85,B 0,C 180,E1 -17839.177,E2 -17839.177} C_VEL
LIN {X 0,Y 282.196,Z 332.381,A -85,B 0,C 180,E1 -17840.595,E2 -17840.595} C_VEL
LIN {X 0,Y 279.992,Z 342.089,A -85,B 0,C 180,E1 -17842.117,E2 -17842.117} C_VEL
LIN {X 0,Y 277.809,Z 351.067,A -85,B 0,C 180,E1 -17843.876,E2 -17843.876} C_VEL
LIN {X 0,Y 275.378,Z 360.172,A -85,B 0,C 180,E1 -17846.105,E2 -17846.105} C_VEL
LIN {X 0,Y 273.51,Z 366.899,A -85,B 0,C 180,E1 -17848.182,E2 -17848.182} C_VEL
LIN {X 0,Y 271.628,Z 373.333,A -85,B 0,C 180,E1 -17850.73,E2 -17850.73} C_VEL
LIN {X 0,Y 270.32,Z 377.853,A -85,B 0,C 180,E1 -17853.091,E2 -17853.091} C_VEL
LIN {X 0,Y 269.125,Z 381.749,A -85,B 0,C 180,E1 -17855.95,E2 -17855.95} C_VEL
LIN {X 0,Y 268.347,Z 384.071,A -85,B 0,C 180,E1 -17858.943,E2 -17858.943} C_VEL
LIN {X 0,Y 268.027,Z 384.748,A -85,B 0,C 180,E1 -17860.959,E2 -17860.959} C_VEL
LIN {X 0,Y 267.836,Z 384.68,A -85,B 0,C 180,E1 -17863.018,E2 -17863.018} C_VEL
LIN {X 0,Y 267.83,Z 383.805,A -85,B 0,C 180,E1 -17865.112,E2 -17865.112} C_VEL
LIN {X 0,Y 267.991,Z 382.101,A -85,B 0,C 180,E1 -17867.247,E2 -17867.247} C_VEL
LIN {X 0,Y 268.265,Z 379.445,A -85,B 0,C 180,E1 -17869.44,E2 -17869.44} C_VEL
LIN {X 0,Y 268.769,Z 375.721,A -85,B 0,C 180,E1 -17871.67,E2 -17871.67} C_VEL
LIN {X 0,Y 269.386,Z 370.673,A -85,B 0,C 180,E1 -17873.974,E2 -17873.974} C_VEL
LIN {X 0,Y 270.194,Z 364.055,A -85,B 0,C 180,E1 -17876.34,E2 -17876.34} C_VEL
LIN {X 0,Y 271.238,Z 357.094,A -85,B 0,C 180,E1 -17878.332,E2 -17878.332} C_VEL
LIN {X 0,Y 272.606,Z 347.859,A -85,B 0,C 180,E1 -17880.459,E2 -17880.459} C_VEL
LIN {X 0,Y 273.971,Z 337.946,A -85,B 0,C 180,E1 -17882.294,E2 -17882.294} C_VEL
LIN {X 0,Y 275.418,Z 327.206,A -85,B 0,C 180,E1 -17883.889,E2 -17883.889} C_VEL
LIN {X 0,Y 276.784,Z 314.824,A -85,B 0,C 180,E1 -17885.325,E2 -17885.325} C_VEL
LIN {X 0,Y 278.04,Z 302.133,A -85,B 0,C 180,E1 -17886.442,E2 -17886.442} C_VEL
LIN {X 0,Y 278.963,Z 288.641,A -85,B 0,C 180,E1 -17887.284,E2 -17887.284} C_VEL
LIN {X 0,Y 279.656,Z 274.841,A -85,B 0,C 180,E1 -17887.831,E2 -17887.831} C_VEL
LIN {X 0,Y 281.768,Z 207.61,A -85,B 0,C 180,E1 -17889.753,E2 -17889.753} C_VEL
LIN {X 0,Y 280.229,Z 199.786,A -85,B 0,C 180,E1 -17890.115,E2 -17890.115} C_VEL
LIN {X 0,Y 271.036,Z 173.45,A -85,B 0,C 180,E1 -17891.725,E2 -17891.725} C_VEL
LIN {X 0,Y 270.328,Z 169.814,A -85,B 0,C 180,E1 -17893.091,E2 -17893.091} C_VEL
LIN {X 0,Y 270.309,Z 169.817,A -85,B 0,C 180,E1 -17896.468,E2 -17896.468} C_VEL
LIN {X 0,Y 270.524,Z 169.784,A -85,B 0,C 180,E1 -17901.033,E2 -17901.033} C_VEL
LIN {X 0,Y 270.506,Z 169.791,A -85,B 0,C 180,E1 -17904.035,E2 -17904.035} C_VEL
LIN {X 0,Y 270.766,Z 169.758,A -85,B 0,C 180,E1 -17908.513,E2 -17908.513} C_VEL
LIN {X 0,Y 270.765,Z 169.758,A -85,B 0,C 180,E1 -17911.488,E2 -17911.488} C_VEL
LIN {X 0,Y 270.559,Z 169.783,A -85,B 0,C 180,E1 -17917.463,E2 -17917.463} C_VEL
LIN {X 0,Y 270.382,Z 169.804,A -85,B 0,C 180,E1 -17920.483,E2 -17920.483} C_VEL
LIN {X 0,Y 270.335,Z 169.81,A -85,B 0,C 180,E1 -17925.069,E2 -17925.069} C_VEL
LIN {X 0,Y 270.216,Z 169.826,A -85,B 0,C 180,E1 -17929.762,E2 -17929.762} C_VEL
LIN {X 0,Y 270.178,Z 169.827,A -85,B 0,C 180,E1 -17934.436,E2 -17934.436} C_VEL
LIN {X 0,Y 270.181,Z 169.829,A -85,B 0,C 180,E1 -17937.919,E2 -17937.919} C_VEL
LIN {X 0,Y 270.165,Z 169.829,A -85,B 0,C 180,E1 -17941.35,E2 -17941.35} C_VEL
LIN {X 0,Y 270.194,Z 169.826,A -85,B 0,C 180,E1 -17944.906,E2 -17944.906} C_VEL
LIN {X 0,Y 270.194,Z 169.827,A -85,B 0,C 180,E1 -17948.711,E2 -17948.711} C_VEL
LIN {X 0,Y 270.143,Z 169.83,A -85,B 0,C 180,E1 -17953.245,E2 -17953.245} C_VEL
LIN {X 0,Y 270.147,Z 169.833,A -85,B 0,C 180,E1 -17957.438,E2 -17957.438} C_VEL
LIN {X 0,Y 270.204,Z 169.825,A -85,B 0,C 180,E1 -17961.374,E2 -17961.374} C_VEL
LIN {X 0,Y 270.194,Z 169.822,A -85,B 0,C 180,E1 -17965.094,E2 -17965.094} C_VEL
LIN {X 0,Y 270.18,Z 169.827,A -85,B 0,C 180,E1 -17969.137,E2 -17969.137} C_VEL
LIN {X 0,Y 270.195,Z 169.826,A -85,B 0,C 180,E1 -17972.173,E2 -17972.173} C_VEL
LIN {X 0,Y 270.178,Z 169.828,A -85,B 0,C 180,E1 -17975.565,E2 -17975.565} C_VEL
LIN {X 0,Y 270.215,Z 169.821,A -85,B 0,C 180,E1 -17980.239,E2 -17980.239} C_VEL
LIN {X 0,Y 270.334,Z 169.807,A -85,B 0,C 180,E1 -17984.932,E2 -17984.932} C_VEL
LIN {X 0,Y 270.38,Z 169.802,A -85,B 0,C 180,E1 -17989.517,E2 -17989.517} C_VEL
LIN {X 0,Y 270.548,Z 169.779,A -85,B 0,C 180,E1 -17992.538,E2 -17992.538} C_VEL
LIN {X 0,Y 270.498,Z 169.785,A -85,B 0,C 180,E1 -17993.887,E2 -17993.887} C_VEL
LIN {X 0,Y 269.879,Z 169.869,A -85,B 0,C 180,E1 -17995.131,E2 -17995.131} C_VEL
LIN {X 0,Y 267.141,Z 170.214,A -85,B 0,C 180,E1 -17997.162,E2 -17997.162} C_VEL
LIN {X 0,Y 264.799,Z 170.503,A -85,B 0,C 180,E1 -17998.812,E2 -17998.812} C_VEL
LIN {X 0,Y 263.789,Z 170.627,A -85,B 0,C 180,E1 -18000.089,E2 -18000.089} C_VEL
LIN {X 0,Y 263.704,Z 170.634,A -85,B 0,C 180,E1 -18000.521,E2 -18000.521} C_VEL
LIN {X 0,Y 263.503,Z 170.658,A -85,B 0,C 180,E1 -18003.058,E2 -18003.058} C_VEL
LIN {X 0,Y 263.511,Z 170.655,A -85,B 0,C 180,E1 -18007.664,E2 -18007.664} C_VEL
LIN {X 0,Y 263.326,Z 170.681,A -85,B 0,C 180,E1 -18010.768,E2 -18010.768} C_VEL
LIN {X 0,Y 263.286,Z 170.688,A -85,B 0,C 180,E1 -18015.483,E2 -18015.483} C_VEL
LIN {X 0,Y 263.205,Z 170.698,A -85,B 0,C 180,E1 -18020.312,E2 -18020.312} C_VEL
LIN {X 0,Y 263.118,Z 170.708,A -85,B 0,C 180,E1 -18025.301,E2 -18025.301} C_VEL
LIN {X 0,Y 263.116,Z 170.709,A -85,B 0,C 180,E1 -18028.738,E2 -18028.738} C_VEL
LIN {X 0,Y 263.125,Z 170.702,A -85,B 0,C 180,E1 -18032.29,E2 -18032.29} C_VEL
LIN {X 0,Y 263.175,Z 170.701,A -85,B 0,C 180,E1 -18036.762,E2 -18036.762} C_VEL
LIN {X 0,Y 263.091,Z 170.711,A -85,B 0,C 180,E1 -18039.876,E2 -18039.876} C_VEL
LIN {X 0,Y 263.076,Z 170.714,A -85,B 0,C 180,E1 -18043.995,E2 -18043.995} C_VEL
LIN {X 0,Y 263.08,Z 170.714,A -85,B 0,C 180,E1 -18048.418,E2 -18048.418} C_VEL
LIN {X 0,Y 263.158,Z 170.704,A -85,B 0,C 180,E1 -18052.103,E2 -18052.103} C_VEL
LIN {X 0,Y 263.198,Z 170.885,A -85,B 0,C 180,E1 -18056.021,E2 -18056.021} C_VEL
LIN {X 0,Y 265.396,Z 181.304,A -85,B 0,C 180,E1 -18059.792,E2 -18059.792} C_VEL
LIN {X 0,Y 266.647,Z 187.74,A -85,B 0,C 180,E1 -18061.961,E2 -18061.961} C_VEL
LIN {X 0,Y 269.788,Z 197.542,A -85,B 0,C 180,E1 -18062.547,E2 -18062.547} C_VEL
LIN {X 0,Y 274.613,Z 233.44,A -85,B 0,C 180,E1 -18064.087,E2 -18064.087} C_VEL
LIN {X 0,Y 272.42,Z 296.556,A -85,B 0,C 180,E1 -18065.975,E2 -18065.975} C_VEL
LIN {X 0,Y 271.448,Z 310.43,A -85,B 0,C 180,E1 -18066.694,E2 -18066.694} C_VEL
LIN {X 0,Y 270.266,Z 322.945,A -85,B 0,C 180,E1 -18067.647,E2 -18067.647} C_VEL
LIN {X 0,Y 268.689,Z 335.358,A -85,B 0,C 180,E1 -18068.921,E2 -18068.921} C_VEL
LIN {X 0,Y 267.147,Z 346.545,A -85,B 0,C 180,E1 -18070.402,E2 -18070.402} C_VEL
LIN {X 0,Y 265.715,Z 357.248,A -85,B 0,C 180,E1 -18072.211,E2 -18072.211} C_VEL
LIN {X 0,Y 264.374,Z 366.655,A -85,B 0,C 180,E1 -18074.188,E2 -18074.188} C_VEL
LIN {X 0,Y 263.28,Z 374.069,A -85,B 0,C 180,E1 -18076.099,E2 -18076.099} C_VEL
LIN {X 0,Y 262.252,Z 381.328,A -85,B 0,C 180,E1 -18078.405,E2 -18078.405} C_VEL
LIN {X 0,Y 261.622,Z 387.09,A -85,B 0,C 180,E1 -18080.725,E2 -18080.725} C_VEL
LIN {X 0,Y 261.257,Z 391.592,A -85,B 0,C 180,E1 -18083.047,E2 -18083.047} C_VEL
LIN {X 0,Y 261.087,Z 394.962,A -85,B 0,C 180,E1 -18085.368,E2 -18085.368} C_VEL
LIN {X 0,Y 261.101,Z 396.622,A -85,B 0,C 180,E1 -18086.914,E2 -18086.914} C_VEL
LIN {X 0,Y 261.12,Z 397.859,A -85,B 0,C 180,E1 -18088.457,E2 -18088.457} C_VEL
LIN {X 0,Y 261.128,Z 398.658,A -85,B 0,C 180,E1 -18090,E2 -18090} C_VEL
LIN {X 0,Y 261.109,Z 399.014,A -85,B 0,C 180,E1 -18091.542,E2 -18091.542} C_VEL
LIN {X 0,Y 261.051,Z 398.971,A -85,B 0,C 180,E1 -18093.086,E2 -18093.086} C_VEL
LIN {X 0,Y 261.087,Z 398.293,A -85,B 0,C 180,E1 -18095.137,E2 -18095.137} C_VEL
LIN {X 0,Y 261.384,Z 396.398,A -85,B 0,C 180,E1 -18097.726,E2 -18097.726} C_VEL
LIN {X 0,Y 261.993,Z 393.7,A -85,B 0,C 180,E1 -18100.041,E2 -18100.041} C_VEL
LIN {X 0,Y 262.928,Z 389.99,A -85,B 0,C 180,E1 -18102.347,E2 -18102.347} C_VEL
LIN {X 0,Y 264.217,Z 385.194,A -85,B 0,C 180,E1 -18104.636,E2 -18104.636} C_VEL
LIN {X 0,Y 266.453,Z 378.018,A -85,B 0,C 180,E1 -18107.261,E2 -18107.261} C_VEL
LIN {X 0,Y 268.387,Z 370.357,A -85,B 0,C 180,E1 -18109.488,E2 -18109.488} C_VEL
LIN {X 0,Y 270.596,Z 362.428,A -85,B 0,C 180,E1 -18111.322,E2 -18111.322} C_VEL
LIN {X 0,Y 273.033,Z 352.878,A -85,B 0,C 180,E1 -18113.112,E2 -18113.112} C_VEL
LIN {X 0,Y 275.564,Z 342.357,A -85,B 0,C 180,E1 -18114.684,E2 -18114.684} C_VEL
LIN {X 0,Y 277.922,Z 330.804,A -85,B 0,C 180,E1 -18116.063,E2 -18116.063} C_VEL
LIN {X 0,Y 280.042,Z 318.656,A -85,B 0,C 180,E1 -18117.157,E2 -18117.157} C_VEL
LIN {X 0,Y 281.934,Z 305.492,A -85,B 0,C 180,E1 -18118.016,E2 -18118.016} C_VEL
LIN {X 0,Y 283.148,Z 292.453,A -85,B 0,C 180,E1 -18118.592,E2 -18118.592} C_VEL
LIN {X 0,Y 286.042,Z 236.34,A -85,B 0,C 180,E1 -18120.264,E2 -18120.264} C_VEL
LIN {X 0,Y 283.919,Z 220.786,A -85,B 0,C 180,E1 -18121.203,E2 -18121.203} C_VEL
LIN {X 0,Y 282.897,Z 215.866,A -85,B 0,C 180,E1 -18121.573,E2 -18121.573} C_VEL
LIN {X 0,Y 277.204,Z 203.049,A -85,B 0,C 180,E1 -18123.116,E2 -18123.116} C_VEL
LIN {X 0,Y 272.278,Z 193.794,A -85,B 0,C 180,E1 -18124.481,E2 -18124.481} C_VEL
LIN {X 0,Y 269.582,Z 189.067,A -85,B 0,C 180,E1 -18125.262,E2 -18125.262} C_VEL
LIN {X 0,Y 267.248,Z 184.669,A -85,B 0,C 180,E1 -18126.035,E2 -18126.035} C_VEL
LIN {X 0,Y 265.249,Z 177.733,A -85,B 0,C 180,E1 -18129.486,E2 -18129.486} C_VEL
LIN {X 0,Y 263.102,Z 170.716,A -85,B 0,C 180,E1 -18133.506,E2 -18133.506} C_VEL
LIN {X 0,Y 263.078,Z 170.711,A -85,B 0,C 180,E1 -18138.097,E2 -18138.097} C_VEL
LIN {X 0,Y 263.145,Z 170.708,A -85,B 0,C 180,E1 -18142.1,E2 -18142.1} C_VEL
LIN {X 0,Y 263.149,Z 170.7,A -85,B 0,C 180,E1 -18145.884,E2 -18145.884} C_VEL
LIN {X 0,Y 263.106,Z 170.703,A -85,B 0,C 180,E1 -18149.5,E2 -18149.5} C_VEL
LIN {X 0,Y 263.11,Z 170.702,A -85,B 0,C 180,E1 -18152.993,E2 -18152.993} C_VEL
LIN {X 0,Y 263.113,Z 170.704,A -85,B 0,C 180,E1 -18156.38,E2 -18156.38} C_VEL
LIN {X 0,Y 263.203,Z 170.699,A -85,B 0,C 180,E1 -18159.688,E2 -18159.688} C_VEL
LIN {X 0,Y 263.283,Z 170.679,A -85,B 0,C 180,E1 -18164.517,E2 -18164.517} C_VEL
LIN {X 0,Y 263.327,Z 170.678,A -85,B 0,C 180,E1 -18169.232,E2 -18169.232} C_VEL
LIN {X 0,Y 263.52,Z 170.653,A -85,B 0,C 180,E1 -18172.336,E2 -18172.336} C_VEL
LIN {X 0,Y 263.727,Z 170.629,A -85,B 0,C 180,E1 -18178.472,E2 -18178.472} C_VEL
LIN {X 0,Y 263.727,Z 170.631,A -85,B 0,C 180,E1 -18181.526,E2 -18181.526} C_VEL
LIN {X 0,Y 263.359,Z 170.813,A -85,B 0,C 180,E1 -18184.687,E2 -18184.687} C_VEL
LIN {X 0,Y 265.046,Z 175.755,A -85,B 0,C 180,E1 -18187.57,E2 -18187.57} C_VEL
LIN {X 0,Y 267.57,Z 179.879,A -85,B 0,C 180,E1 -18188.353,E2 -18188.353} C_VEL
LIN {X 0,Y 273.945,Z 190.323,A -85,B 0,C 180,E1 -18190.191,E2 -18190.191} C_VEL
LIN {X 0,Y 279.675,Z 200.875,A -85,B 0,C 180,E1 -18191.731,E2 -18191.731} C_VEL
LIN {X 0,Y 284.828,Z 211.895,A -85,B 0,C 180,E1 -18193.084,E2 -18193.084} C_VEL
LIN {X 0,Y 286.934,Z 217.087,A -85,B 0,C 180,E1 -18193.628,E2 -18193.628} C_VEL
LIN {X 0,Y 283.322,Z 283.548,A -85,B 0,C 180,E1 -18195.621,E2 -18195.621} C_VEL
LIN {X 0,Y 281.994,Z 296.769,A -85,B 0,C 180,E1 -18196.282,E2 -18196.282} C_VEL
LIN {X 0,Y 280.581,Z 308.142,A -85,B 0,C 180,E1 -18197.116,E2 -18197.116} C_VEL
LIN {X 0,Y 278.769,Z 319.273,A -85,B 0,C 180,E1 -18198.178,E2 -18198.178} C_VEL
LIN {X 0,Y 276.461,Z 330.546,A -85,B 0,C 180,E1 -18199.556,E2 -18199.556} C_VEL
LIN {X 0,Y 274.044,Z 341.125,A -85,B 0,C 180,E1 -18201.199,E2 -18201.199} C_VEL
LIN {X 0,Y 271.888,Z 349.553,A -85,B 0,C 180,E1 -18202.813,E2 -18202.813} C_VEL
LIN {X 0,Y 269.782,Z 357.319,A -85,B 0,C 180,E1 -18204.633,E2 -18204.633} C_VEL
LIN {X 0,Y 267.321,Z 365.559,A -85,B 0,C 180,E1 -18207.057,E2 -18207.057} C_VEL
LIN {X 0,Y 265.249,Z 372.36,A -85,B 0,C 180,E1 -18209.652,E2 -18209.652} C_VEL
LIN {X 0,Y 263.677,Z 377.402,A -85,B 0,C 180,E1 -18212.213,E2 -18212.213} C_VEL
LIN {X 0,Y 262.328,Z 381.507,A -85,B 0,C 180,E1 -18215.169,E2 -18215.169} C_VEL
LIN {X 0,Y 261.4,Z 384.061,A -85,B 0,C 180,E1 -18218.197,E2 -18218.197} C_VEL
LIN {X 0,Y 260.923,Z 384.979,A -85,B 0,C 180,E1 -18221.047,E2 -18221.047} C_VEL
LIN {X 0,Y 260.731,Z 384.745,A -85,B 0,C 180,E1 -18223.3,E2 -18223.3} C_VEL
LIN {X 0,Y 260.743,Z 383.682,A -85,B 0,C 180,E1 -18225.51,E2 -18225.51} C_VEL
LIN {X 0,Y 260.953,Z 381.788,A -85,B 0,C 180,E1 -18227.679,E2 -18227.679} C_VEL
LIN {X 0,Y 261.381,Z 377.945,A -85,B 0,C 180,E1 -18230.541,E2 -18230.541} C_VEL
LIN {X 0,Y 261.953,Z 373.833,A -85,B 0,C 180,E1 -18232.758,E2 -18232.758} C_VEL
LIN {X 0,Y 262.709,Z 367.564,A -85,B 0,C 180,E1 -18235.357,E2 -18235.357} C_VEL
LIN {X 0,Y 263.836,Z 359.962,A -85,B 0,C 180,E1 -18237.809,E2 -18237.809} C_VEL
LIN {X 0,Y 265.152,Z 351.219,A -85,B 0,C 180,E1 -18240.031,E2 -18240.031} C_VEL
LIN {X 0,Y 266.617,Z 341.244,A -85,B 0,C 180,E1 -18242.068,E2 -18242.068} C_VEL
LIN {X 0,Y 268.073,Z 330.926,A -85,B 0,C 180,E1 -18243.743,E2 -18243.743} C_VEL
LIN {X 0,Y 269.555,Z 318.479,A -85,B 0,C 180,E1 -18245.345,E2 -18245.345} C_VEL
LIN {X 0,Y 270.826,Z 306.892,A -85,B 0,C 180,E1 -18246.486,E2 -18246.486} C_VEL
LIN {X 0,Y 271.901,Z 293.059,A -85,B 0,C 180,E1 -18247.49,E2 -18247.49} C_VEL
LIN {X 0,Y 272.669,Z 280.38,A -85,B 0,C 180,E1 -18248.107,E2 -18248.107} C_VEL
LIN {X 0,Y 275.131,Z 208.648,A -85,B 0,C 180,E1 -18250.23,E2 -18250.23} C_VEL
LIN {X 0,Y 273.759,Z 201.843,A -85,B 0,C 180,E1 -18250.553,E2 -18250.553} C_VEL
LIN {X 0,Y 263.848,Z 173.647,A -85,B 0,C 180,E1 -18252.333,E2 -18252.333} C_VEL
LIN {X 0,Y 263.264,Z 170.694,A -85,B 0,C 180,E1 -18253.553,E2 -18253.553} C_VEL
LIN {X 0,Y 263.292,Z 170.69,A -85,B 0,C 180,E1 -18257.67,E2 -18257.67} C_VEL
LIN {X 0,Y 263.469,Z 170.664,A -85,B 0,C 180,E1 -18260.791,E2 -18260.791} C_VEL
LIN {X 0,Y 263.478,Z 170.665,A -85,B 0,C 180,E1 -18263.875,E2 -18263.875} C_VEL
LIN {X 0,Y 263.73,Z 170.635,A -85,B 0,C 180,E1 -18268.473,E2 -18268.473} C_VEL
LIN {X 0,Y 263.728,Z 170.635,A -85,B 0,C 180,E1 -18271.527,E2 -18271.527} C_VEL
LIN {X 0,Y 263.523,Z 170.661,A -85,B 0,C 180,E1 -18277.663,E2 -18277.663} C_VEL
LIN {X 0,Y 263.327,Z 170.683,A -85,B 0,C 180,E1 -18280.768,E2 -18280.768} C_VEL
LIN {X 0,Y 263.285,Z 170.69,A -85,B 0,C 180,E1 -18285.482,E2 -18285.482} C_VEL
LIN {X 0,Y 263.204,Z 170.696,A -85,B 0,C 180,E1 -18290.311,E2 -18290.311} C_VEL
LIN {X 0,Y 263.116,Z 170.71,A -85,B 0,C 180,E1 -18295.301,E2 -18295.301} C_VEL
LIN {X 0,Y 263.114,Z 170.708,A -85,B 0,C 180,E1 -18298.737,E2 -18298.737} C_VEL
LIN {X 0,Y 263.123,Z 170.702,A -85,B 0,C 180,E1 -18302.289,E2 -18302.289} C_VEL
LIN {X 0,Y 263.172,Z 170.702,A -85,B 0,C 180,E1 -18306.761,E2 -18306.761} C_VEL
LIN {X 0,Y 263.087,Z 170.71,A -85,B 0,C 180,E1 -18309.875,E2 -18309.875} C_VEL
LIN {X 0,Y 263.072,Z 170.707,A -85,B 0,C 180,E1 -18313.994,E2 -18313.994} C_VEL
LIN {X 0,Y 263.076,Z 170.713,A -85,B 0,C 180,E1 -18318.418,E2 -18318.418} C_VEL
LIN {X 0,Y 263.153,Z 170.702,A -85,B 0,C 180,E1 -18322.103,E2 -18322.103} C_VEL
LIN {X 0,Y 263.148,Z 170.696,A -85,B 0,C 180,E1 -18325.886,E2 -18325.886} C_VEL
LIN {X 0,Y 263.122,Z 170.704,A -85,B 0,C 180,E1 -18329.504,E2 -18329.504} C_VEL
LIN {X 0,Y 263.122,Z 170.709,A -85,B 0,C 180,E1 -18332.996,E2 -18332.996} C_VEL
LIN {X 0,Y 263.111,Z 170.711,A -85,B 0,C 180,E1 -18336.381,E2 -18336.381} C_VEL
LIN {X 0,Y 263.203,Z 170.691,A -85,B 0,C 180,E1 -18339.689,E2 -18339.689} C_VEL
LIN {X 0,Y 263.284,Z 170.687,A -85,B 0,C 180,E1 -18344.519,E2 -18344.519} C_VEL
LIN {X 0,Y 263.325,Z 170.68,A -85,B 0,C 180,E1 -18349.233,E2 -18349.233} C_VEL
LIN {X 0,Y 263.51,Z 170.657,A -85,B 0,C 180,E1 -18352.337,E2 -18352.337} C_VEL
LIN {X 0,Y 263.727,Z 170.632,A -85,B 0,C 180,E1 -18358.474,E2 -18358.474} C_VEL
LIN {X 0,Y 263.704,Z 170.634,A -85,B 0,C 180,E1 -18360.521,E2 -18360.521} C_VEL
LIN {X 0,Y 263.002,Z 170.724,A -85,B 0,C 180,E1 -18361.793,E2 -18361.793} C_VEL
LIN {X 0,Y 260.046,Z 171.093,A -85,B 0,C 180,E1 -18363.861,E2 -18363.861} C_VEL
LIN {X 0,Y 257.554,Z 171.399,A -85,B 0,C 180,E1 -18365.544,E2 -18365.544} C_VEL
LIN {X 0,Y 256.503,Z 171.524,A -85,B 0,C 180,E1 -18366.852,E2 -18366.852} C_VEL
LIN {X 0,Y 256.428,Z 171.534,A -85,B 0,C 180,E1 -18367.296,E2 -18367.296} C_VEL
LIN {X 0,Y 256.27,Z 171.56,A -85,B 0,C 180,E1 -18371.068,E2 -18371.068} C_VEL
LIN {X 0,Y 256.21,Z 171.566,A -85,B 0,C 180,E1 -18375.921,E2 -18375.921} C_VEL
LIN {X 0,Y 256.117,Z 171.582,A -85,B 0,C 180,E1 -18381.097,E2 -18381.097} C_VEL
LIN {X 0,Y 256.08,Z 171.583,A -85,B 0,C 180,E1 -18385.088,E2 -18385.088} C_VEL
LIN {X 0,Y 256.075,Z 171.586,A -85,B 0,C 180,E1 -18388.57,E2 -18388.57} C_VEL
LIN {X 0,Y 256.069,Z 171.582,A -85,B 0,C 180,E1 -18391.7,E2 -18391.7} C_VEL
LIN {X 0,Y 256.079,Z 171.582,A -85,B 0,C 180,E1 -18395.194,E2 -18395.194} C_VEL
LIN {X 0,Y 256.11,Z 171.584,A -85,B 0,C 180,E1 -18397.27,E2 -18397.27} C_VEL
LIN {X 0,Y 256.018,Z 171.597,A -85,B 0,C 180,E1 -18401.211,E2 -18401.211} C_VEL
LIN {X 0,Y 256.018,Z 171.594,A -85,B 0,C 180,E1 -18405.54,E2 -18405.54} C_VEL
LIN {X 0,Y 256.019,Z 171.596,A -85,B 0,C 180,E1 -18408.79,E2 -18408.79} C_VEL
LIN {X 0,Y 256.127,Z 171.583,A -85,B 0,C 180,E1 -18412.867,E2 -18412.867} C_VEL
LIN {X 0,Y 256.128,Z 171.65,A -85,B 0,C 180,E1 -18415.551,E2 -18415.551} C_VEL
LIN {X 0,Y 258.477,Z 182.815,A -85,B 0,C 180,E1 -18419.707,E2 -18419.707} C_VEL
LIN {X 0,Y 259.381,Z 187.514,A -85,B 0,C 180,E1 -18421.324,E2 -18421.324} C_VEL
LIN {X 0,Y 263.349,Z 199.965,A -85,B 0,C 180,E1 -18422.094,E2 -18422.094} C_VEL
LIN {X 0,Y 267.844,Z 232.935,A -85,B 0,C 180,E1 -18423.562,E2 -18423.562} C_VEL
LIN {X 0,Y 265.687,Z 295.505,A -85,B 0,C 180,E1 -18425.483,E2 -18425.483} C_VEL
LIN {X 0,Y 264.791,Z 308.899,A -85,B 0,C 180,E1 -18426.176,E2 -18426.176} C_VEL
LIN {X 0,Y 263.581,Z 321.824,A -85,B 0,C 180,E1 -18427.152,E2 -18427.152} C_VEL
LIN {X 0,Y 262.064,Z 333.646,A -85,B 0,C 180,E1 -18428.362,E2 -18428.362} C_VEL
LIN {X 0,Y 260.48,Z 345.112,A -85,B 0,C 180,E1 -18429.879,E2 -18429.879} C_VEL
LIN {X 0,Y 259.059,Z 354.829,A -85,B 0,C 180,E1 -18431.488,E2 -18431.488} C_VEL
LIN {X 0,Y 257.808,Z 364.012,A -85,B 0,C 180,E1 -18433.367,E2 -18433.367} C_VEL
LIN {X 0,Y 256.355,Z 373.215,A -85,B 0,C 180,E1 -18435.716,E2 -18435.716} C_VEL
LIN {X 0,Y 255.251,Z 380.615,A -85,B 0,C 180,E1 -18438.082,E2 -18438.082} C_VEL
LIN {X 0,Y 254.579,Z 386.504,A -85,B 0,C 180,E1 -18440.466,E2 -18440.466} C_VEL
LIN {X 0,Y 254.178,Z 391.098,A -85,B 0,C 180,E1 -18442.852,E2 -18442.852} C_VEL
LIN {X 0,Y 254.016,Z 394.554,A -85,B 0,C 180,E1 -18445.239,E2 -18445.239} C_VEL
LIN {X 0,Y 254.016,Z 396.254,A -85,B 0,C 180,E1 -18446.828,E2 -18446.828} C_VEL
LIN {X 0,Y 254.049,Z 397.531,A -85,B 0,C 180,E1 -18448.415,E2 -18448.415} C_VEL
LIN {X 0,Y 254.056,Z 398.392,A -85,B 0,C 180,E1 -18450,E2 -18450} C_VEL
LIN {X 0,Y 254.015,Z 398.796,A -85,B 0,C 180,E1 -18451.585,E2 -18451.585} C_VEL
LIN {X 0,Y 253.95,Z 398.79,A -85,B 0,C 180,E1 -18453.173,E2 -18453.173} C_VEL
LIN {X 0,Y 253.992,Z 398.295,A -85,B 0,C 180,E1 -18455.038,E2 -18455.038} C_VEL
LIN {X 0,Y 254.337,Z 396.365,A -85,B 0,C 180,E1 -18457.941,E2 -18457.941} C_VEL
LIN {X 0,Y 254.987,Z 393.758,A -85,B 0,C 180,E1 -18460.32,E2 -18460.32} C_VEL
LIN {X 0,Y 255.963,Z 390.147,A -85,B 0,C 180,E1 -18462.688,E2 -18462.688} C_VEL
LIN {X 0,Y 257.353,Z 385.442,A -85,B 0,C 180,E1 -18465.036,E2 -18465.036} C_VEL
LIN {X 0,Y 259.698,Z 378.364,A -85,B 0,C 180,E1 -18467.724,E2 -18467.724} C_VEL
LIN {X 0,Y 261.651,Z 371.099,A -85,B 0,C 180,E1 -18469.929,E2 -18469.929} C_VEL
LIN {X 0,Y 264.041,Z 363.076,A -85,B 0,C 180,E1 -18471.878,E2 -18471.878} C_VEL
LIN {X 0,Y 266.575,Z 353.792,A -85,B 0,C 180,E1 -18473.706,E2 -18473.706} C_VEL
LIN {X 0,Y 269.496,Z 342.273,A -85,B 0,C 180,E1 -18475.485,E2 -18475.485} C_VEL
LIN {X 0,Y 271.977,Z 330.751,A -85,B 0,C 180,E1 -18476.885,E2 -18476.885} C_VEL
LIN {X 0,Y 274.197,Z 318.644,A -85,B 0,C 180,E1 -18477.993,E2 -18477.993} C_VEL
LIN {X 0,Y 276.146,Z 305.557,A -85,B 0,C 180,E1 -18478.865,E2 -18478.865} C_VEL
LIN {X 0,Y 277.446,Z 292.668,A -85,B 0,C 180,E1 -18479.447,E2 -18479.447} C_VEL
LIN {X 0,Y 280.437,Z 237.329,A -85,B 0,C 180,E1 -18481.14,E2 -18481.14} C_VEL
LIN {X 0,Y 278.553,Z 222.861,A -85,B 0,C 180,E1 -18482.053,E2 -18482.053} C_VEL
LIN {X 0,Y 277.749,Z 218.992,A -85,B 0,C 180,E1 -18482.357,E2 -18482.357} C_VEL
LIN {X 0,Y 272.459,Z 206.999,A -85,B 0,C 180,E1 -18483.862,E2 -18483.862} C_VEL
LIN {X 0,Y 267.769,Z 198.059,A -85,B 0,C 180,E1 -18485.244,E2 -18485.244} C_VEL
LIN {X 0,Y 262.77,Z 189.213,A -85,B 0,C 180,E1 -18486.8,E2 -18486.8} C_VEL
LIN {X 0,Y 260.12,Z 184.767,A -85,B 0,C 180,E1 -18487.679,E2 -18487.679} C_VEL
LIN {X 0,Y 259.252,Z 182.029,A -85,B 0,C 180,E1 -18489.005,E2 -18489.005} C_VEL
LIN {X 0,Y 257.34,Z 175.902,A -85,B 0,C 180,E1 -18492.491,E2 -18492.491} C_VEL
LIN {X 0,Y 256.008,Z 171.594,A -85,B 0,C 180,E1 -18495.312,E2 -18495.312} C_VEL
LIN {X 0,Y 256.017,Z 171.595,A -85,B 0,C 180,E1 -18498.788,E2 -18498.788} C_VEL
LIN {X 0,Y 256.119,Z 171.575,A -85,B 0,C 180,E1 -18502.865,E2 -18502.865} C_VEL
LIN {X 0,Y 256.063,Z 171.579,A -85,B 0,C 180,E1 -18506.706,E2 -18506.706} C_VEL
LIN {X 0,Y 256.038,Z 171.581,A -85,B 0,C 180,E1 -18510.39,E2 -18510.39} C_VEL
LIN {X 0,Y 256.064,Z 171.577,A -85,B 0,C 180,E1 -18513.95,E2 -18513.95} C_VEL
LIN {X 0,Y 256.054,Z 171.578,A -85,B 0,C 180,E1 -18517.401,E2 -18517.401} C_VEL
LIN {X 0,Y 256.1,Z 171.574,A -85,B 0,C 180,E1 -18520.772,E2 -18520.772} C_VEL
LIN {X 0,Y 256.208,Z 171.563,A -85,B 0,C 180,E1 -18524.079,E2 -18524.079} C_VEL
LIN {X 0,Y 256.271,Z 171.555,A -85,B 0,C 180,E1 -18528.932,E2 -18528.932} C_VEL
LIN {X 0,Y 256.463,Z 171.531,A -85,B 0,C 180,E1 -18532.124,E2 -18532.124} C_VEL
LIN {X 0,Y 256.443,Z 171.543,A -85,B 0,C 180,E1 -18536.857,E2 -18536.857} C_VEL
LIN {X 0,Y 256.689,Z 171.506,A -85,B 0,C 180,E1 -18538.43,E2 -18538.43} C_VEL
LIN {X 0,Y 256.689,Z 171.508,A -85,B 0,C 180,E1 -18541.568,E2 -18541.568} C_VEL
LIN {X 0,Y 256.508,Z 171.613,A -85,B 0,C 180,E1 -18542.944,E2 -18542.944} C_VEL
LIN {X 0,Y 257.814,Z 176.153,A -85,B 0,C 180,E1 -18545.769,E2 -18545.769} C_VEL
LIN {X 0,Y 260.809,Z 180.584,A -85,B 0,C 180,E1 -18546.769,E2 -18546.769} C_VEL
LIN {X 0,Y 264.804,Z 186.873,A -85,B 0,C 180,E1 -18548.057,E2 -18548.057} C_VEL
LIN {X 0,Y 271.569,Z 198.299,A -85,B 0,C 180,E1 -18550.054,E2 -18550.054} C_VEL
LIN {X 0,Y 278.1,Z 211.424,A -85,B 0,C 180,E1 -18551.878,E2 -18551.878} C_VEL
LIN {X 0,Y 281.359,Z 219.24,A -85,B 0,C 180,E1 -18552.778,E2 -18552.778} C_VEL
LIN {X 0,Y 277.649,Z 283.608,A -85,B 0,C 180,E1 -18554.753,E2 -18554.753} C_VEL
LIN {X 0,Y 276.286,Z 296.674,A -85,B 0,C 180,E1 -18555.411,E2 -18555.411} C_VEL
LIN {X 0,Y 274.641,Z 309.22,A -85,B 0,C 180,E1 -18556.348,E2 -18556.348} C_VEL
LIN {X 0,Y 272.623,Z 320.637,A -85,B 0,C 180,E1 -18557.482,E2 -18557.482} C_VEL
LIN {X 0,Y 270.099,Z 332.363,A -85,B 0,C 180,E1 -18558.98,E2 -18558.98} C_VEL
LIN {X 0,Y 267.732,Z 342.079,A -85,B 0,C 180,E1 -18560.554,E2 -18560.554} C_VEL
LIN {X 0,Y 265.28,Z 351.024,A -85,B 0,C 180,E1 -18562.353,E2 -18562.353} C_VEL
LIN {X 0,Y 262.669,Z 359.707,A -85,B 0,C 180,E1 -18564.538,E2 -18564.538} C_VEL
LIN {X 0,Y 260.252,Z 367.403,A -85,B 0,C 180,E1 -18566.984,E2 -18566.984} C_VEL
LIN {X 0,Y 258.261,Z 373.388,A -85,B 0,C 180,E1 -18569.449,E2 -18569.449} C_VEL
LIN {X 0,Y 256.713,Z 377.989,A -85,B 0,C 180,E1 -18571.933,E2 -18571.933} C_VEL
LIN {X 0,Y 255.54,Z 381.357,A -85,B 0,C 180,E1 -18574.406,E2 -18574.406} C_VEL
LIN {X 0,Y 254.484,Z 384.008,A -85,B 0,C 180,E1 -18577.413,E2 -18577.413} C_VEL
LIN {X 0,Y 254.054,Z 384.949,A -85,B 0,C 180,E1 -18579.512,E2 -18579.512} C_VEL
LIN {X 0,Y 253.741,Z 385.21,A -85,B 0,C 180,E1 -18581.661,E2 -18581.661} C_VEL
LIN {X 0,Y 253.613,Z 384.678,A -85,B 0,C 180,E1 -18583.906,E2 -18583.906} C_VEL
LIN {X 0,Y 253.678,Z 383.291,A -85,B 0,C 180,E1 -18586.164,E2 -18586.164} C_VEL
LIN {X 0,Y 253.946,Z 381.105,A -85,B 0,C 180,E1 -18588.38,E2 -18588.38} C_VEL
LIN {X 0,Y 254.308,Z 377.891,A -85,B 0,C 180,E1 -18590.695,E2 -18590.695} C_VEL
LIN {X 0,Y 254.921,Z 373.473,A -85,B 0,C 180,E1 -18593.082,E2 -18593.082} C_VEL
LIN {X 0,Y 255.668,Z 367.582,A -85,B 0,C 180,E1 -18595.553,E2 -18595.553} C_VEL
LIN {X 0,Y 256.823,Z 360.068,A -85,B 0,C 180,E1 -18598.028,E2 -18598.028} C_VEL
LIN {X 0,Y 258.066,Z 351.945,A -85,B 0,C 180,E1 -18600.159,E2 -18600.159} C_VEL
LIN {X 0,Y 259.475,Z 342.611,A -85,B 0,C 180,E1 -18602.146,E2 -18602.146} C_VEL
LIN {X 0,Y 260.931,Z 332.85,A -85,B 0,C 180,E1 -18603.83,E2 -18603.83} C_VEL
LIN {X 0,Y 262.394,Z 321.626,A -85,B 0,C 180,E1 -18605.377,E2 -18605.377} C_VEL
LIN {X 0,Y 263.802,Z 308.87,A -85,B 0,C 180,E1 -18606.74,E2 -18606.74} C_VEL
LIN {X 0,Y 264.908,Z 296.269,A -85,B 0,C 180,E1 -18607.737,E2 -18607.737} C_VEL
LIN {X 0,Y 265.789,Z 282.535,A -85,B 0,C 180,E1 -18608.479,E2 -18608.479} C_VEL
LIN {X 0,Y 267.82,Z 228.925,A -85,B 0,C 180,E1 -18610.129,E2 -18610.129} C_VEL
LIN {X 0,Y 268.39,Z 208.958,A -85,B 0,C 180,E1 -18610.745,E2 -18610.745} C_VEL
LIN {X 0,Y 267.149,Z 203.507,A -85,B 0,C 180,E1 -18611.026,E2 -18611.026} C_VEL
LIN {X 0,Y 257.506,Z 176.293,A -85,B 0,C 180,E1 -18612.79,E2 -18612.79} C_VEL
LIN {X 0,Y 256.664,Z 173.85,A -85,B 0,C 180,E1 -18612.985,E2 -18612.985} C_VEL
LIN {X 0,Y 256.237,Z 171.571,A -85,B 0,C 180,E1 -18613.975,E2 -18613.975} C_VEL
LIN {X 0,Y 256.27,Z 171.563,A -85,B 0,C 180,E1 -18618.933,E2 -18618.933} C_VEL
LIN {X 0,Y 256.465,Z 171.539,A -85,B 0,C 180,E1 -18622.125,E2 -18622.125} C_VEL
LIN {X 0,Y 256.447,Z 171.54,A -85,B 0,C 180,E1 -18626.858,E2 -18626.858} C_VEL
LIN {X 0,Y 256.692,Z 171.512,A -85,B 0,C 180,E1 -18628.431,E2 -18628.431} C_VEL
LIN {X 0,Y 256.691,Z 171.512,A -85,B 0,C 180,E1 -18631.569,E2 -18631.569} C_VEL
LIN {X 0,Y 256.45,Z 171.542,A -85,B 0,C 180,E1 -18636.294,E2 -18636.294} C_VEL
LIN {X 0,Y 256.399,Z 171.548,A -85,B 0,C 180,E1 -18639.466,E2 -18639.466} C_VEL
LIN {X 0,Y 256.198,Z 171.572,A -85,B 0,C 180,E1 -18644.293,E2 -18644.293} C_VEL
LIN {X 0,Y 256.144,Z 171.579,A -85,B 0,C 180,E1 -18647.567,E2 -18647.567} C_VEL
LIN {X 0,Y 256.116,Z 171.58,A -85,B 0,C 180,E1 -18651.097,E2 -18651.097} C_VEL
LIN {X 0,Y 256.079,Z 171.585,A -85,B 0,C 180,E1 -18655.087,E2 -18655.087} C_VEL
LIN {X 0,Y 256.072,Z 171.585,A -85,B 0,C 180,E1 -18658.569,E2 -18658.569} C_VEL
LIN {X 0,Y 256.066,Z 171.583,A -85,B 0,C 180,E1 -18661.7,E2 -18661.7} C_VEL
LIN {X 0,Y 256.076,Z 171.587,A -85,B 0,C 180,E1 -18665.194,E2 -18665.194} C_VEL
LIN {X 0,Y 256.107,Z 171.585,A -85,B 0,C 180,E1 -18667.269,E2 -18667.269} C_VEL
LIN {X 0,Y 256.014,Z 171.591,A -85,B 0,C 180,E1 -18671.211,E2 -18671.211} C_VEL
LIN {X 0,Y 256.013,Z 171.591,A -85,B 0,C 180,E1 -18675.54,E2 -18675.54} C_VEL
LIN {X 0,Y 256.014,Z 171.595,A -85,B 0,C 180,E1 -18678.79,E2 -18678.79} C_VEL
LIN {X 0,Y 256.121,Z 171.58,A -85,B 0,C 180,E1 -18682.867,E2 -18682.867} C_VEL
LIN {X 0,Y 256.062,Z 171.58,A -85,B 0,C 180,E1 -18686.707,E2 -18686.707} C_VEL
LIN {X 0,Y 256.05,Z 171.586,A -85,B 0,C 180,E1 -18690.393,E2 -18690.393} C_VEL
LIN {X 0,Y 256.07,Z 171.586,A -85,B 0,C 180,E1 -18693.952,E2 -18693.952} C_VEL
LIN {X 0,Y 256.053,Z 171.585,A -85,B 0,C 180,E1 -18697.403,E2 -18697.403} C_VEL
LIN {X 0,Y 256.102,Z 171.572,A -85,B 0,C 180,E1 -18700.774,E2 -18700.774} C_VEL
LIN {X 0,Y 256.209,Z 171.564,A -85,B 0,C 180,E1 -18704.08,E2 -18704.08} C_VEL
LIN {X 0,Y 256.269,Z 171.56,A -85,B 0,C 180,E1 -18708.933,E2 -18708.933} C_VEL
LIN {X 0,Y 256.452,Z 171.538,A -85,B 0,C 180,E1 -18712.125,E2 -18712.125} C_VEL
LIN {X 0,Y 256.439,Z 171.535,A -85,B 0,C 180,E1 -18716.859,E2 -18716.859} C_VEL
LIN {X 0,Y 256.69,Z 171.508,A -85,B 0,C 180,E1 -18718.432,E2 -18718.432} C_VEL
LIN {X 0,Y 256.69,Z 171.509,A -85,B 0,C 180,E1 -18721.57,E2 -18721.57} C_VEL
LIN {X 0,Y 256.428,Z 171.534,A -85,B 0,C 180,E1 -18727.296,E2 -18727.296} C_VEL
LIN {X 0,Y 255.755,Z 171.624,A -85,B 0,C 180,E1 -18728.605,E2 -18728.605} C_VEL
LIN {X 0,Y 252.791,Z 171.994,A -85,B 0,C 180,E1 -18730.735,E2 -18730.735} C_VEL
LIN {X 0,Y 250.271,Z 172.308,A -85,B 0,C 180,E1 -18732.47,E2 -18732.47} C_VEL
LIN {X 0,Y 249.205,Z 172.443,A -85,B 0,C 180,E1 -18733.819,E2 -18733.819} C_VEL
LIN {X 0,Y 249.128,Z 172.447,A -85,B 0,C 180,E1 -18734.277,E2 -18734.277} C_VEL
LIN {X 0,Y 249.075,Z 172.457,A -85,B 0,C 180,E1 -18738.083,E2 -18738.083} C_VEL
LIN {X 0,Y 249.041,Z 172.466,A -85,B 0,C 180,E1 -18741.523,E2 -18741.523} C_VEL
LIN {X 0,Y 249.042,Z 172.462,A -85,B 0,C 180,E1 -18745.44,E2 -18745.44} C_VEL
LIN {X 0,Y 249.023,Z 172.466,A -85,B 0,C 180,E1 -18748.969,E2 -18748.969} C_VEL
LIN {X 0,Y 249.025,Z 172.457,A -85,B 0,C 180,E1 -18752.427,E2 -18752.427} C_VEL
LIN {X 0,Y 249.026,Z 172.462,A -85,B 0,C 180,E1 -18756.347,E2 -18756.347} C_VEL
LIN {X 0,Y 248.979,Z 172.469,A -85,B 0,C 180,E1 -18760.484,E2 -18760.484} C_VEL
LIN {X 0,Y 248.962,Z 172.475,A -85,B 0,C 180,E1 -18764.889,E2 -18764.889} C_VEL
LIN {X 0,Y 248.979,Z 172.471,A -85,B 0,C 180,E1 -18767.355,E2 -18767.355} C_VEL
LIN {X 0,Y 249.041,Z 172.463,A -85,B 0,C 180,E1 -18772.202,E2 -18772.202} C_VEL
LIN {X 0,Y 249.086,Z 172.544,A -85,B 0,C 180,E1 -18775.114,E2 -18775.114} C_VEL
LIN {X 0,Y 251.379,Z 183.522,A -85,B 0,C 180,E1 -18779.321,E2 -18779.321} C_VEL
LIN {X 0,Y 252.092,Z 187.107,A -85,B 0,C 180,E1 -18780.65,E2 -18780.65} C_VEL
LIN {X 0,Y 256.848,Z 201.654,A -85,B 0,C 180,E1 -18781.593,E2 -18781.593} C_VEL
LIN {X 0,Y 261.187,Z 234.191,A -85,B 0,C 180,E1 -18783.083,E2 -18783.083} C_VEL
LIN {X 0,Y 258.93,Z 295.482,A -85,B 0,C 180,E1 -18785.014,E2 -18785.014} C_VEL
LIN {X 0,Y 257.944,Z 309.542,A -85,B 0,C 180,E1 -18785.77,E2 -18785.77} C_VEL
LIN {X 0,Y 256.762,Z 321.702,A -85,B 0,C 180,E1 -18786.723,E2 -18786.723} C_VEL
LIN {X 0,Y 255.203,Z 333.505,A -85,B 0,C 180,E1 -18787.962,E2 -18787.962} C_VEL
LIN {X 0,Y 253.582,Z 344.965,A -85,B 0,C 180,E1 -18789.519,E2 -18789.519} C_VEL
LIN {X 0,Y 252.02,Z 355.348,A -85,B 0,C 180,E1 -18791.296,E2 -18791.296} C_VEL
LIN {X 0,Y 250.68,Z 364.682,A -85,B 0,C 180,E1 -18793.3,E2 -18793.3} C_VEL
LIN {X 0,Y 249.236,Z 373.748,A -85,B 0,C 180,E1 -18795.716,E2 -18795.716} C_VEL
LIN {X 0,Y 248.12,Z 380.992,A -85,B 0,C 180,E1 -18798.15,E2 -18798.15} C_VEL
LIN {X 0,Y 247.384,Z 387.574,A -85,B 0,C 180,E1 -18801.011,E2 -18801.011} C_VEL
LIN {X 0,Y 247.06,Z 391.875,A -85,B 0,C 180,E1 -18803.466,E2 -18803.466} C_VEL
LIN {X 0,Y 246.924,Z 394.134,A -85,B 0,C 180,E1 -18805.102,E2 -18805.102} C_VEL
LIN {X 0,Y 246.916,Z 395.885,A -85,B 0,C 180,E1 -18806.736,E2 -18806.736} C_VEL
LIN {X 0,Y 246.957,Z 397.202,A -85,B 0,C 180,E1 -18808.369,E2 -18808.369} C_VEL
LIN {X 0,Y 246.985,Z 398.104,A -85,B 0,C 180,E1 -18810,E2 -18810} C_VEL
LIN {X 0,Y 246.922,Z 398.577,A -85,B 0,C 180,E1 -18811.631,E2 -18811.631} C_VEL
LIN {X 0,Y 246.854,Z 398.609,A -85,B 0,C 180,E1 -18813.264,E2 -18813.264} C_VEL
LIN {X 0,Y 246.884,Z 398.25,A -85,B 0,C 180,E1 -18814.899,E2 -18814.899} C_VEL
LIN {X 0,Y 247.015,Z 397.501,A -85,B 0,C 180,E1 -18816.534,E2 -18816.534} C_VEL
LIN {X 0,Y 247.287,Z 396.348,A -85,B 0,C 180,E1 -18818.169,E2 -18818.169} C_VEL
LIN {X 0,Y 247.973,Z 393.812,A -85,B 0,C 180,E1 -18820.615,E2 -18820.615} C_VEL
LIN {X 0,Y 249.007,Z 390.276,A -85,B 0,C 180,E1 -18823.049,E2 -18823.049} C_VEL
LIN {X 0,Y 250.507,Z 385.665,A -85,B 0,C 180,E1 -18825.457,E2 -18825.457} C_VEL
LIN {X 0,Y 252.959,Z 378.744,A -85,B 0,C 180,E1 -18828.213,E2 -18828.213} C_VEL
LIN {X 0,Y 254.96,Z 371.852,A -85,B 0,C 180,E1 -18830.409,E2 -18830.409} C_VEL
LIN {X 0,Y 257.515,Z 363.77,A -85,B 0,C 180,E1 -18832.462,E2 -18832.462} C_VEL
LIN {X 0,Y 260.148,Z 354.697,A -85,B 0,C 180,E1 -18834.329,E2 -18834.329} C_VEL
LIN {X 0,Y 262.894,Z 344.727,A -85,B 0,C 180,E1 -18835.96,E2 -18835.96} C_VEL
LIN {X 0,Y 265.394,Z 333.801,A -85,B 0,C 180,E1 -18837.394,E2 -18837.394} C_VEL
LIN {X 0,Y 267.881,Z 321.748,A -85,B 0,C 180,E1 -18838.606,E2 -18838.606} C_VEL
LIN {X 0,Y 269.95,Z 309.316,A -85,B 0,C 180,E1 -18839.539,E2 -18839.539} C_VEL
LIN {X 0,Y 271.578,Z 295.489,A -85,B 0,C 180,E1 -18840.252,E2 -18840.252} C_VEL
LIN {X 0,Y 274.322,Z 250.611,A -85,B 0,C 180,E1 -18841.67,E2 -18841.67} C_VEL
LIN {X 0,Y 274.932,Z 237.731,A -85,B 0,C 180,E1 -18842.091,E2 -18842.091} C_VEL
LIN {X 0,Y 272.944,Z 222.878,A -85,B 0,C 180,E1 -18843.084,E2 -18843.084} C_VEL
LIN {X 0,Y 267.982,Z 211.351,A -85,B 0,C 180,E1 -18844.595,E2 -18844.595} C_VEL
LIN {X 0,Y 263.288,Z 202.246,A -85,B 0,C 180,E1 -18846.043,E2 -18846.043} C_VEL
LIN {X 0,Y 258.748,Z 194.049,A -85,B 0,C 180,E1 -18847.552,E2 -18847.552} C_VEL
LIN {X 0,Y 255.556,Z 188.9,A -85,B 0,C 180,E1 -18848.647,E2 -18848.647} C_VEL
LIN {X 0,Y 252.902,Z 184.727,A -85,B 0,C 180,E1 -18849.618,E2 -18849.618} C_VEL
LIN {X 0,Y 252.6,Z 184.005,A -85,B 0,C 180,E1 -18849.785,E2 -18849.785} C_VEL
LIN {X 0,Y 250.828,Z 178.24,A -85,B 0,C 180,E1 -18853.238,E2 -18853.238} C_VEL
LIN {X 0,Y 248.972,Z 172.468,A -85,B 0,C 180,E1 -18857.284,E2 -18857.284} C_VEL
LIN {X 0,Y 249.018,Z 172.466,A -85,B 0,C 180,E1 -18861.617,E2 -18861.617} C_VEL
LIN {X 0,Y 249.04,Z 172.459,A -85,B 0,C 180,E1 -18865.638,E2 -18865.638} C_VEL
LIN {X 0,Y 248.991,Z 172.46,A -85,B 0,C 180,E1 -18869.464,E2 -18869.464} C_VEL
LIN {X 0,Y 249.011,Z 172.457,A -85,B 0,C 180,E1 -18873.154,E2 -18873.154} C_VEL
LIN {X 0,Y 249.003,Z 172.459,A -85,B 0,C 180,E1 -18876.724,E2 -18876.724} C_VEL
LIN {X 0,Y 249.037,Z 172.457,A -85,B 0,C 180,E1 -18880.205,E2 -18880.205} C_VEL
LIN {X 0,Y 249.154,Z 172.445,A -85,B 0,C 180,E1 -18883.615,E2 -18883.615} C_VEL
LIN {X 0,Y 249.216,Z 172.432,A -85,B 0,C 180,E1 -18888.614,E2 -18888.614} C_VEL
LIN {X 0,Y 249.409,Z 172.409,A -85,B 0,C 180,E1 -18891.9,E2 -18891.9} C_VEL
LIN {X 0,Y 249.252,Z 172.429,A -85,B 0,C 180,E1 -18895.147,E2 -18895.147} C_VEL
LIN {X 0,Y 249.651,Z 172.382,A -85,B 0,C 180,E1 -18898.386,E2 -18898.386} C_VEL
LIN {X 0,Y 249.648,Z 172.482,A -85,B 0,C 180,E1 -18901.007,E2 -18901.007} C_VEL
LIN {X 0,Y 250.58,Z 176.565,A -85,B 0,C 180,E1 -18903.718,E2 -18903.718} C_VEL
LIN {X 0,Y 253.499,Z 180.857,A -85,B 0,C 180,E1 -18904.827,E2 -18904.827} C_VEL
LIN {X 0,Y 255.07,Z 182.891,A -85,B 0,C 180,E1 -18905.384,E2 -18905.384} C_VEL
LIN {X 0,Y 258.55,Z 188.13,A -85,B 0,C 180,E1 -18906.582,E2 -18906.582} C_VEL
LIN {X 0,Y 261.727,Z 193.359,A -85,B 0,C 180,E1 -18907.639,E2 -18907.639} C_VEL
LIN {X 0,Y 267.4,Z 203.129,A -85,B 0,C 180,E1 -18909.392,E2 -18909.392} C_VEL
LIN {X 0,Y 273.778,Z 216.432,A -85,B 0,C 180,E1 -18911.287,E2 -18911.287} C_VEL
LIN {X 0,Y 275.862,Z 221.755,A -85,B 0,C 180,E1 -18911.898,E2 -18911.898} C_VEL
LIN {X 0,Y 272.07,Z 284.05,A -85,B 0,C 180,E1 -18913.847,E2 -18913.847} C_VEL
LIN {X 0,Y 270.563,Z 297.582,A -85,B 0,C 180,E1 -18914.55,E2 -18914.55} C_VEL
LIN {X 0,Y 268.885,Z 309.486,A -85,B 0,C 180,E1 -18915.465,E2 -18915.465} C_VEL
LIN {X 0,Y 266.526,Z 321.999,A -85,B 0,C 180,E1 -18916.752,E2 -18916.752} C_VEL
LIN {X 0,Y 263.829,Z 333.89,A -85,B 0,C 180,E1 -18918.338,E2 -18918.338} C_VEL
LIN {X 0,Y 261.092,Z 344.202,A -85,B 0,C 180,E1 -18920.105,E2 -18920.105} C_VEL
LIN {X 0,Y 258.679,Z 352.471,A -85,B 0,C 180,E1 -18921.864,E2 -18921.864} C_VEL
LIN {X 0,Y 256.236,Z 360.136,A -85,B 0,C 180,E1 -18923.863,E2 -18923.863} C_VEL
LIN {X 0,Y 253.704,Z 367.622,A -85,B 0,C 180,E1 -18926.309,E2 -18926.309} C_VEL
LIN {X 0,Y 251.459,Z 373.956,A -85,B 0,C 180,E1 -18929.022,E2 -18929.022} C_VEL
LIN {X 0,Y 249.949,Z 378.072,A -85,B 0,C 180,E1 -18931.307,E2 -18931.307} C_VEL
LIN {X 0,Y 248.43,Z 382.137,A -85,B 0,C 180,E1 -18934.456,E2 -18934.456} C_VEL
LIN {X 0,Y 247.436,Z 384.405,A -85,B 0,C 180,E1 -18937.319,E2 -18937.319} C_VEL
LIN {X 0,Y 246.908,Z 385.318,A -85,B 0,C 180,E1 -18939.78,E2 -18939.78} C_VEL
